LIN {X 0,Y 124.094,Z 764.223,A -85,B 0,C 180,E1 27360.319,E2 27360.319} C_VEL
LIN {X 0,Y 133.281,Z 757.884,A -85,B 0,C 180,E1 27361.4,E2 27361.4} C_VEL
LIN {X 0,Y 134.55,Z 756.801,A -85,B 0,C 180,E1 27362,E2 27362} C_VEL
LIN {X 0,Y 132.092,Z 757.455,A -85,B 0,C 180,E1 27366.547,E2 27366.547} C_VEL
LIN {X 0,Y 129.508,Z 758.725,A -85,B 0,C 180,E1 27369.46,E2 27369.46} C_VEL
LIN {X 0,Y 123.075,Z 762.693,A -85,B 0,C 180,E1 27371.274,E2 27371.274} C_VEL
LIN {X 0,Y 91.987,Z 778.369,A -85,B 0,C 180,E1 27378.553,E2 27378.553} C_VEL
LIN {X 0,Y 62.704,Z 788.454,A -85,B 0,C 180,E1 27392.644,E2 27392.644} C_VEL
LIN {X 0,Y 40.148,Z 793.378,A -85,B 0,C 180,E1 27427.943,E2 27427.943} C_VEL
LIN {X 0,Y 40.207,Z 793.347,A -85,B 0,C 180,E1 27472.061,E2 27472.061} C_VEL
LIN {X 0,Y 62.756,Z 788.368,A -85,B 0,C 180,E1 27507.325,E2 27507.325} C_VEL
LIN {X 0,Y 92.44,Z 778.051,A -85,B 0,C 180,E1 27521.5,E2 27521.5} C_VEL
LIN {X 0,Y 124.79,Z 761.469,A -85,B 0,C 180,E1 27528.95,E2 27528.95} C_VEL
LIN {X 0,Y 129.483,Z 758.548,A -85,B 0,C 180,E1 27530.56,E2 27530.56} C_VEL
LIN {X 0,Y 132.115,Z 757.233,A -85,B 0,C 180,E1 27533.454,E2 27533.454} C_VEL
LIN {X 0,Y 134.548,Z 756.597,A -85,B 0,C 180,E1 27538.001,E2 27538.001} C_VEL
LIN {X 0,Y 126.384,Z 762.482,A -85,B 0,C 180,E1 27539.383,E2 27539.383} C_VEL
LIN {X 0,Y 94.415,Z 781.112,A -85,B 0,C 180,E1 27544.833,E2 27544.833} C_VEL
LIN {X 0,Y 63.041,Z 794.367,A -85,B 0,C 180,E1 27556.741,E2 27556.741} C_VEL
LIN {X 0,Y 40.652,Z 801.7,A -85,B 0,C 180,E1 27582.041,E2 27582.041} C_VEL
LIN {X 0,Y 34.452,Z 804.774,A -85,B 0,C 180,E1 27629.345,E2 27629.345} C_VEL
LIN {X 0,Y 34.228,Z 804.663,A -85,B 0,C 180,E1 27643.351,E2 27643.351} C_VEL
LIN {X 0,Y 35.461,Z 800.565,A -85,B 0,C 180,E1 27687.235,E2 27687.235} C_VEL
LIN {X 0,Y 36.191,Z 800.352,A -85,B 0,C 180,E1 27688.651,E2 27688.651} C_VEL
LIN {X 0,Y 65.88,Z 791.602,A -85,B 0,C 180,E1 27712.667,E2 27712.667} C_VEL
LIN {X 0,Y 98.193,Z 777.913,A -85,B 0,C 180,E1 27720.886,E2 27720.886} C_VEL
LIN {X 0,Y 126.325,Z 761.604,A -85,B 0,C 180,E1 27724.614,E2 27724.614} C_VEL
LIN {X 0,Y 124.467,Z 762.35,A -85,B 0,C 180,E1 27726.95,E2 27726.95} C_VEL
LIN {X 0,Y 92.927,Z 778.287,A -85,B 0,C 180,E1 27733.062,E2 27733.062} C_VEL
LIN {X 0,Y 65.374,Z 787.866,A -85,B 0,C 180,E1 27742.624,E2 27742.624} C_VEL
LIN {X 0,Y 41.377,Z 793.304,A -85,B 0,C 180,E1 27763.193,E2 27763.193} C_VEL
LIN {X 0,Y 29.353,Z 795.095,A -85,B 0,C 180,E1 27810.025,E2 27810.025} C_VEL
LIN {X 0,Y 41.486,Z 793.244,A -85,B 0,C 180,E1 27856.698,E2 27856.698} C_VEL
LIN {X 0,Y 72.099,Z 785.77,A -85,B 0,C 180,E1 27880.383,E2 27880.383} C_VEL
LIN {X 0,Y 103.697,Z 773.349,A -85,B 0,C 180,E1 27889.212,E2 27889.212} C_VEL
LIN {X 0,Y 124.456,Z 762.164,A -85,B 0,C 180,E1 27893.05,E2 27893.05} C_VEL
LIN {X 0,Y 126.367,Z 761.386,A -85,B 0,C 180,E1 27895.382,E2 27895.382} C_VEL
LIN {X 0,Y 95.503,Z 779.134,A -85,B 0,C 180,E1 27899.572,E2 27899.572} C_VEL
LIN {X 0,Y 61.185,Z 793.12,A -85,B 0,C 180,E1 27909.364,E2 27909.364} C_VEL
LIN {X 0,Y 35.694,Z 800.457,A -85,B 0,C 180,E1 27932.24,E2 27932.24} C_VEL
LIN {X 0,Y 26.54,Z 803.586,A -85,B 0,C 180,E1 27989.973,E2 27989.973} C_VEL
LIN {X 0,Y 36.191,Z 800.352,A -85,B 0,C 180,E1 28048.651,E2 28048.651} C_VEL
LIN {X 0,Y 46.867,Z 796.623,A -85,B 0,C 180,E1 28067.322,E2 28067.322} C_VEL
LIN {X 0,Y 60.341,Z 791.95,A -85,B 0,C 180,E1 28078.38,E2 28078.38} C_VEL
LIN {X 0,Y 95.606,Z 778.16,A -85,B 0,C 180,E1 28085.323,E2 28085.323} C_VEL
LIN {X 0,Y 103.062,Z 774.499,A -85,B 0,C 180,E1 28086.079,E2 28086.079} C_VEL
LIN {X 0,Y 69.826,Z 787.065,A -85,B 0,C 180,E1 28093.53,E2 28093.53} C_VEL
LIN {X 0,Y 36.478,Z 794.49,A -85,B 0,C 180,E1 28114.212,E2 28114.212} C_VEL
LIN {X 0,Y 21.544,Z 796.282,A -85,B 0,C 180,E1 28170.034,E2 28170.034} C_VEL
LIN {X 0,Y 36.571,Z 794.431,A -85,B 0,C 180,E1 28225.644,E2 28225.644} C_VEL
LIN {X 0,Y 69.863,Z 786.962,A -85,B 0,C 180,E1 28246.435,E2 28246.435} C_VEL
LIN {X 0,Y 103.212,Z 774.29,A -85,B 0,C 180,E1 28253.914,E2 28253.914} C_VEL
LIN {X 0,Y 70.179,Z 788.574,A -85,B 0,C 180,E1 28258.944,E2 28258.944} C_VEL
LIN {X 0,Y 37.396,Z 798.04,A -85,B 0,C 180,E1 28273.988,E2 28273.988} C_VEL
LIN {X 0,Y 21.421,Z 801.316,A -85,B 0,C 180,E1 28305.17,E2 28305.17} C_VEL
LIN {X 0,Y 18.54,Z 802.371,A -85,B 0,C 180,E1 28349.961,E2 28349.961} C_VEL
LIN {X 0,Y 32.056,Z 799.249,A -85,B 0,C 180,E1 28420.225,E2 28420.225} C_VEL
LIN {X 0,Y 60.341,Z 791.95,A -85,B 0,C 180,E1 28438.38,E2 28438.38} C_VEL
LIN {X 0,Y 59.231,Z 791.67,A -85,B 0,C 180,E1 28442.189,E2 28442.189} C_VEL
LIN {X 0,Y 53.428,Z 792.556,A -85,B 0,C 180,E1 28446.947,E2 28446.947} C_VEL
LIN {X 0,Y 34.694,Z 795.461,A -85,B 0,C 180,E1 28461.032,E2 28461.032} C_VEL
LIN {X 0,Y 31.971,Z 795.746,A -85,B 0,C 180,E1 28463.533,E2 28463.533} C_VEL
LIN {X 0,Y 13.763,Z 797.464,A -85,B 0,C 180,E1 28530.053,E2 28530.053} C_VEL
LIN {X 0,Y 32.797,Z 795.62,A -85,B 0,C 180,E1 28597.006,E2 28597.006} C_VEL
LIN {X 0,Y 61.116,Z 790.16,A -85,B 0,C 180,E1 28611.036,E2 28611.036} C_VEL
LIN {X 0,Y 65.791,Z 789.027,A -85,B 0,C 180,E1 28612.984,E2 28612.984} C_VEL
LIN {X 0,Y 30.308,Z 797.97,A -85,B 0,C 180,E1 28625.039,E2 28625.039} C_VEL
LIN {X 0,Y 10.527,Z 801.154,A -85,B 0,C 180,E1 28709.931,E2 28709.931} C_VEL
LIN {X 0,Y 30.282,Z 798.006,A -85,B 0,C 180,E1 28794.973,E2 28794.973} C_VEL
LIN {X 0,Y 65.728,Z 789.134,A -85,B 0,C 180,E1 28807.007,E2 28807.007} C_VEL
LIN {X 0,Y 39.585,Z 794.659,A -85,B 0,C 180,E1 28817.704,E2 28817.704} C_VEL
LIN {X 0,Y 31.971,Z 795.746,A -85,B 0,C 180,E1 28823.533,E2 28823.533} C_VEL
LIN {X 0,Y 24.943,Z 796.903,A -85,B 0,C 180,E1 28824.135,E2 28824.135} C_VEL
LIN {X 0,Y 11.311,Z 799.26,A -85,B 0,C 180,E1 28801.153,E2 28801.153} C_VEL
LIN {X 0,Y 9.86,Z 799.371,A -85,B 0,C 180,E1 28798.609,E2 28798.609} C_VEL
LIN {X 0,Y 2.505,Z 799.935,A -85,B 0,C 180,E1 28709.709,E2 28709.709} C_VEL
LIN {X 0,Y 23.792,Z 797.786,A -85,B 0,C 180,E1 28611.393,E2 28611.393} C_VEL
LIN {X 0,Y 20.158,Z 797.842,A -85,B 0,C 180,E1 28603.349,E2 28603.349} C_VEL
LIN {X 0,Y 16.218,Z 798.123,A -85,B 0,C 180,E1 28461.626,E2 28461.626} C_VEL
LIN {X 0,Y 23.673,Z 797.839,A -85,B 0,C 180,E1 28448.557,E2 28448.557} C_VEL
LIN {X 0,Y 9.86,Z 799.371,A -85,B 0,C 180,E1 28438.609,E2 28438.609} C_VEL
LIN {X 0,Y 8.044,Z 801.368,A -85,B 0,C 180,E1 28435.281,E2 28435.281} C_VEL
LIN {X 0,Y 8.044,Z 875,A -85,B 0,C 180,E1 28435.281,E2 28435.281} C_VEL
LIN {X 0,Y 8.044,Z 875,A -85,B 0,C 180,E1 28435.281,E2 28435.281}

QRS_NEXT_CUT()
PTP {E1 28256.944,E2 28256.944}
PTP {X 0,Y 607.85,A -85,B 0,C 180,E1 28256.944,E2 28256.944,E3 0,E4 0,E5 0,E6 0}
QRS_SPEED_INIT()
LIN {X 0,Y 607.85,Z 875,A -85,B 0,C 180,E1 28256.944,E2 28256.944,E3 0,E4 0,E5 0,E6 0} C_VEL
LIN {X 0,Y 607.85,Z 296.842,A -85,B 0,C 180,E1 28256.944,E2 28256.944} C_VEL
LIN {X 0,Y 607.85,Z 288.764,A -85,B 0,C 180,E1 28256.944,E2 28256.944} C_VEL
LIN {X 0,Y 607.871,Z 286.764,A -85,B 0,C 180,E1 28256.755,E2 28256.755} C_VEL
LIN {X 0,Y 607.835,Z 286.764,A -85,B 0,C 180,E1 28253.672,E2 28253.672} C_VEL
LIN {X 0,Y 607.851,Z 286.764,A -85,B 0,C 180,E1 28250.914,E2 28250.914} C_VEL
LIN {X 0,Y 607.842,Z 286.764,A -85,B 0,C 180,E1 28247.652,E2 28247.652} C_VEL
LIN {X 0,Y 607.86,Z 286.764,A -85,B 0,C 180,E1 28244.839,E2 28244.839} C_VEL
LIN {X 0,Y 607.85,Z 286.762,A -85,B 0,C 180,E1 28241.589,E2 28241.589} C_VEL
LIN {X 0,Y 607.875,Z 286.764,A -85,B 0,C 180,E1 28238.684,E2 28238.684} C_VEL
LIN {X 0,Y 607.856,Z 286.761,A -85,B 0,C 180,E1 28235.511,E2 28235.511} C_VEL
LIN {X 0,Y 607.886,Z 286.764,A -85,B 0,C 180,E1 28232.577,E2 28232.577} C_VEL
LIN {X 0,Y 607.862,Z 286.761,A -85,B 0,C 180,E1 28229.451,E2 28229.451} C_VEL
LIN {X 0,Y 607.899,Z 286.764,A -85,B 0,C 180,E1 28226.451,E2 28226.451} C_VEL
LIN {X 0,Y 607.865,Z 286.76,A -85,B 0,C 180,E1 28223.338,E2 28223.338} C_VEL
LIN {X 0,Y 607.909,Z 286.765,A -85,B 0,C 180,E1 28220.329,E2 28220.329} C_VEL
LIN {X 0,Y 607.867,Z 286.76,A -85,B 0,C 180,E1 28217.188,E2 28217.188} C_VEL
LIN {X 0,Y 607.915,Z 286.761,A -85,B 0,C 180,E1 28214.083,E2 28214.083} C_VEL
LIN {X 0,Y 607.87,Z 286.76,A -85,B 0,C 180,E1 28210.975,E2 28210.975} C_VEL
LIN {X 0,Y 607.912,Z 286.759,A -85,B 0,C 180,E1 28207.841,E2 28207.841} C_VEL
LIN {X 0,Y 607.879,Z 286.761,A -85,B 0,C 180,E1 28204.687,E2 28204.687} C_VEL
LIN {X 0,Y 607.911,Z 286.755,A -85,B 0,C 180,E1 28201.535,E2 28201.535} C_VEL
LIN {X 0,Y 607.905,Z 286.765,A -85,B 0,C 180,E1 28198.273,E2 28198.273} C_VEL
LIN {X 0,Y 607.909,Z 287.028,A -85,B 0,C 180,E1 28196.259,E2 28196.259} C_VEL
LIN {X 0,Y 607.912,Z 319.926,A -85,B 0,C 180,E1 28193.454,E2 28193.454} C_VEL
LIN {X 0,Y 607.914,Z 334.281,A -85,B 0,C 180,E1 28192.278,E2 28192.278} C_VEL
LIN {X 0,Y 607.916,Z 541.958,A -85,B 0,C 180,E1 28189.666,E2 28189.666} C_VEL
LIN {X 0,Y 607.911,Z 560.928,A -85,B 0,C 180,E1 28189.25,E2 28189.25} C_VEL
LIN {X 0,Y 607.902,Z 579.266,A -85,B 0,C 180,E1 28188.668,E2 28188.668} C_VEL
LIN {X 0,Y 607.897,Z 597.163,A -85,B 0,C 180,E1 28187.913,E2 28187.913} C_VEL
LIN {X 0,Y 607.919,Z 613.869,A -85,B 0,C 180,E1 28187.023,E2 28187.023} C_VEL
LIN {X 0,Y 607.917,Z 629.704,A -85,B 0,C 180,E1 28185.991,E2 28185.991} C_VEL
LIN {X 0,Y 607.917,Z 644.611,A -85,B 0,C 180,E1 28184.818,E2 28184.818} C_VEL
LIN {X 0,Y 607.915,Z 658.52,A -85,B 0,C 180,E1 28183.506,E2 28183.506} C_VEL
LIN {X 0,Y 607.917,Z 671.323,A -85,B 0,C 180,E1 28182.056,E2 28182.056} C_VEL
LIN {X 0,Y 607.911,Z 682.566,A -85,B 0,C 180,E1 28180.519,E2 28180.519} C_VEL
LIN {X 0,Y 607.914,Z 692.264,A -85,B 0,C 180,E1 28178.894,E2 28178.894} C_VEL
LIN {X 0,Y 607.911,Z 699.987,A -85,B 0,C 180,E1 28177.276,E2 28177.276} C_VEL
LIN {X 0,Y 607.907,Z 706.267,A -85,B 0,C 180,E1 28175.569,E2 28175.569} C_VEL
LIN {X 0,Y 607.918,Z 710.775,A -85,B 0,C 180,E1 28173.867,E2 28173.867} C_VEL
LIN {X 0,Y 607.917,Z 713.734,A -85,B 0,C 180,E1 28172.074,E2 28172.074} C_VEL
LIN {X 0,Y 607.908,Z 714.929,A -85,B 0,C 180,E1 28170.283,E2 28170.283} C_VEL
LIN {X 0,Y 607.915,Z 714.38,A -85,B 0,C 180,E1 28168.492,E2 28168.492} C_VEL
LIN {X 0,Y 607.909,Z 712.08,A -85,B 0,C 180,E1 28166.7,E2 28166.7} C_VEL
LIN {X 0,Y 607.914,Z 708.217,A -85,B 0,C 180,E1 28164.999,E2 28164.999} C_VEL
LIN {X 0,Y 607.91,Z 702.635,A -85,B 0,C 180,E1 28163.294,E2 28163.294} C_VEL
LIN {X 0,Y 607.917,Z 695.641,A -85,B 0,C 180,E1 28161.678,E2 28161.678} C_VEL
LIN {X 0,Y 607.913,Z 686.781,A -85,B 0,C 180,E1 28160.056,E2 28160.056} C_VEL
LIN {X 0,Y 607.917,Z 676.477,A -85,B 0,C 180,E1 28158.521,E2 28158.521} C_VEL
LIN {X 0,Y 607.913,Z 664.743,A -85,B 0,C 180,E1 28157.075,E2 28157.075} C_VEL
LIN {X 0,Y 607.917,Z 651.561,A -85,B 0,C 180,E1 28155.718,E2 28155.718} C_VEL
LIN {X 0,Y 607.917,Z 636.801,A -85,B 0,C 180,E1 28154.45,E2 28154.45} C_VEL
LIN {X 0,Y 607.917,Z 620.944,A -85,B 0,C 180,E1 28153.322,E2 28153.322} C_VEL
LIN {X 0,Y 607.902,Z 603.949,A -85,B 0,C 180,E1 28152.335,E2 28152.335} C_VEL
LIN {X 0,Y 607.918,Z 586.961,A -85,B 0,C 180,E1 28151.543,E2 28151.543} C_VEL
LIN {X 0,Y 607.909,Z 569.084,A -85,B 0,C 180,E1 28150.895,E2 28150.895} C_VEL
LIN {X 0,Y 607.915,Z 550.763,A -85,B 0,C 180,E1 28150.413,E2 28150.413} C_VEL
LIN {X 0,Y 607.918,Z 531.813,A -85,B 0,C 180,E1 28150.096,E2 28150.096} C_VEL
LIN {X 0,Y 607.91,Z 334.059,A -85,B 0,C 180,E1 28147.621,E2 28147.621} C_VEL
LIN {X 0,Y 607.918,Z 296.429,A -85,B 0,C 180,E1 28144.475,E2 28144.475} C_VEL
LIN {X 0,Y 607.909,Z 286.947,A -85,B 0,C 180,E1 28143.636,E2 28143.636} C_VEL
LIN {X 0,Y 607.91,Z 286.756,A -85,B 0,C 180,E1 28140.543,E2 28140.543} C_VEL
LIN {X 0,Y 607.889,Z 286.762,A -85,B 0,C 180,E1 28137.352,E2 28137.352} C_VEL
LIN {X 0,Y 607.91,Z 286.758,A -85,B 0,C 180,E1 28134.181,E2 28134.181} C_VEL
LIN {X 0,Y 607.877,Z 286.76,A -85,B 0,C 180,E1 28131.075,E2 28131.075} C_VEL
LIN {X 0,Y 607.91,Z 286.76,A -85,B 0,C 180,E1 28127.98,E2 28127.98} C_VEL
LIN {X 0,Y 607.872,Z 286.759,A -85,B 0,C 180,E1 28124.882,E2 28124.882} C_VEL
LIN {X 0,Y 607.918,Z 286.764,A -85,B 0,C 180,E1 28121.696,E2 28121.696} C_VEL
LIN {X 0,Y 607.877,Z 286.759,A -85,B 0,C 180,E1 28118.565,E2 28118.565} C_VEL
LIN {X 0,Y 607.879,Z 286.763,A -85,B 0,C 180,E1 28115.264,E2 28115.264} C_VEL
LIN {X 0,Y 607.897,Z 286.758,A -85,B 0,C 180,E1 28112.203,E2 28112.203} C_VEL
LIN {X 0,Y 607.862,Z 286.762,A -85,B 0,C 180,E1 28109.028,E2 28109.028} C_VEL
LIN {X 0,Y 607.903,Z 286.759,A -85,B 0,C 180,E1 28106.05,E2 28106.05} C_VEL
LIN {X 0,Y 607.854,Z 286.763,A -85,B 0,C 180,E1 28102.91,E2 28102.91} C_VEL
LIN {X 0,Y 607.905,Z 286.76,A -85,B 0,C 180,E1 28099.905,E2 28099.905} C_VEL
LIN {X 0,Y 607.846,Z 286.763,A -85,B 0,C 180,E1 28096.801,E2 28096.801} C_VEL
LIN {X 0,Y 607.909,Z 286.761,A -85,B 0,C 180,E1 28093.798,E2 28093.798} C_VEL
LIN {X 0,Y 607.839,Z 286.764,A -85,B 0,C 180,E1 28090.713,E2 28090.713} C_VEL
LIN {X 0,Y 607.899,Z 286.762,A -85,B 0,C 180,E1 28087.751,E2 28087.751} C_VEL
LIN {X 0,Y 607.834,Z 286.764,A -85,B 0,C 180,E1 28084.718,E2 28084.718} C_VEL
LIN {X 0,Y 607.866,Z 286.764,A -85,B 0,C 180,E1 28081.885,E2 28081.885} C_VEL
LIN {X 0,Y 607.834,Z 286.765,A -85,B 0,C 180,E1 28078.775,E2 28078.775} C_VEL
LIN {X 0,Y 607.846,Z 286.764,A -85,B 0,C 180,E1 28076.039,E2 28076.039} C_VEL
LIN {X 0,Y 607.848,Z 286.763,A -85,B 0,C 180,E1 28072.819,E2 28072.819} C_VEL
LIN {X 0,Y 607.847,Z 286.764,A -85,B 0,C 180,E1 28070.054,E2 28070.054} C_VEL
LIN {X 0,Y 607.857,Z 286.762,A -85,B 0,C 180,E1 28066.783,E2 28066.783} C_VEL
LIN {X 0,Y 607.856,Z 286.764,A -85,B 0,C 180,E1 28063.958,E2 28063.958} C_VEL
LIN {X 0,Y 607.861,Z 286.761,A -85,B 0,C 180,E1 28060.694,E2 28060.694} C_VEL
LIN {X 0,Y 607.873,Z 286.764,A -85,B 0,C 180,E1 28057.771,E2 28057.771} C_VEL
LIN {X 0,Y 607.862,Z 286.761,A -85,B 0,C 180,E1 28054.557,E2 28054.557} C_VEL
LIN {X 0,Y 607.889,Z 286.764,A -85,B 0,C 180,E1 28051.618,E2 28051.618} C_VEL
LIN {X 0,Y 607.865,Z 286.76,A -85,B 0,C 180,E1 28048.432,E2 28048.432} C_VEL
LIN {X 0,Y 607.918,Z 286.763,A -85,B 0,C 180,E1 28045.314,E2 28045.314} C_VEL
LIN {X 0,Y 607.867,Z 286.76,A -85,B 0,C 180,E1 28042.274,E2 28042.274} C_VEL
LIN {X 0,Y 607.914,Z 286.761,A -85,B 0,C 180,E1 28039.162,E2 28039.162} C_VEL
LIN {X 0,Y 607.871,Z 286.76,A -85,B 0,C 180,E1 28036.042,E2 28036.042} C_VEL
LIN {X 0,Y 607.913,Z 286.759,A -85,B 0,C 180,E1 28032.914,E2 28032.914} C_VEL
LIN {X 0,Y 607.88,Z 286.761,A -85,B 0,C 180,E1 28029.778,E2 28029.778} C_VEL
LIN {X 0,Y 607.908,Z 286.756,A -85,B 0,C 180,E1 28026.54,E2 28026.54} C_VEL
LIN {X 0,Y 607.897,Z 286.884,A -85,B 0,C 180,E1 28023.498,E2 28023.498} C_VEL
LIN {X 0,Y 607.908,Z 287.709,A -85,B 0,C 180,E1 28023.382,E2 28023.382} C_VEL
LIN {X 0,Y 607.913,Z 340.141,A -85,B 0,C 180,E1 28020.435,E2 28020.435} C_VEL
LIN {X 0,Y 607.885,Z 390.509,A -85,B 0,C 180,E1 28017.701,E2 28017.701} C_VEL
LIN {X 0,Y 607.913,Z 616.116,A -85,B 0,C 180,E1 28014.784,E2 28014.784} C_VEL
LIN {X 0,Y 607.918,Z 653.733,A -85,B 0,C 180,E1 28014.278,E2 28014.278} C_VEL
LIN {X 0,Y 607.906,Z 673.698,A -85,B 0,C 180,E1 28013.84,E2 28013.84} C_VEL
LIN {X 0,Y 607.911,Z 693.06,A -85,B 0,C 180,E1 28013.249,E2 28013.249} C_VEL
LIN {X 0,Y 607.915,Z 712.501,A -85,B 0,C 180,E1 28012.482,E2 28012.482} C_VEL
LIN {X 0,Y 607.919,Z 731.168,A -85,B 0,C 180,E1 28011.567,E2 28011.567} C_VEL
LIN {X 0,Y 607.917,Z 749.766,A -85,B 0,C 180,E1 28010.456,E2 28010.456} C_VEL
LIN {X 0,Y 607.913,Z 767.254,A -85,B 0,C 180,E1 28009.204,E2 28009.204} C_VEL
LIN {X 0,Y 607.911,Z 783.162,A -85,B 0,C 180,E1 28007.863,E2 28007.863} C_VEL
LIN {X 0,Y 607.915,Z 797.673,A -85,B 0,C 180,E1 28006.432,E2 28006.432} C_VEL
LIN {X 0,Y 607.909,Z 811.263,A -85,B 0,C 180,E1 28004.867,E2 28004.867} C_VEL
LIN {X 0,Y 607.918,Z 823.719,A -85,B 0,C 180,E1 28003.176,E2 28003.176} C_VEL
LIN {X 0,Y 607.906,Z 834.252,A -85,B 0,C 180,E1 28001.479,E2 28001.479} C_VEL
LIN {X 0,Y 607.907,Z 843.561,A -85,B 0,C 180,E1 27999.658,E2 27999.658} C_VEL
LIN {X 0,Y 607.907,Z 850.973,A -85,B 0,C 180,E1 27997.846,E2 27997.846} C_VEL
LIN {X 0,Y 607.913,Z 856.989,A -85,B 0,C 180,E1 27995.947,E2 27995.947} C_VEL
LIN {X 0,Y 607.913,Z 861.292,A -85,B 0,C 180,E1 27994.055,E2 27994.055} C_VEL
LIN {X 0,Y 607.909,Z 863.95,A -85,B 0,C 180,E1 27992.168,E2 27992.168} C_VEL
LIN {X 0,Y 607.902,Z 864.94,A -85,B 0,C 180,E1 27990.283,E2 27990.283} C_VEL
LIN {X 0,Y 607.904,Z 864.372,A -85,B 0,C 180,E1 27988.398,E2 27988.398} C_VEL
LIN {X 0,Y 607.908,Z 862.082,A -85,B 0,C 180,E1 27986.417,E2 27986.417} C_VEL
LIN {X 0,Y 607.91,Z 858.255,A -85,B 0,C 180,E1 27984.526,E2 27984.526} C_VEL
LIN {X 0,Y 607.913,Z 852.689,A -85,B 0,C 180,E1 27982.629,E2 27982.629} C_VEL
LIN {X 0,Y 607.919,Z 845.655,A -85,B 0,C 180,E1 27980.82,E2 27980.82} C_VEL
LIN {X 0,Y 607.909,Z 836.843,A -85,B 0,C 180,E1 27979.001,E2 27979.001} C_VEL
LIN {X 0,Y 607.911,Z 826.516,A -85,B 0,C 180,E1 27977.247,E2 27977.247} C_VEL
LIN {X 0,Y 607.917,Z 815.136,A -85,B 0,C 180,E1 27975.62,E2 27975.62} C_VEL
LIN {X 0,Y 607.91,Z 801.355,A -85,B 0,C 180,E1 27973.96,E2 27973.96} C_VEL
LIN {X 0,Y 607.918,Z 785.904,A -85,B 0,C 180,E1 27972.385,E2 27972.385} C_VEL
LIN {X 0,Y 607.913,Z 769.201,A -85,B 0,C 180,E1 27970.945,E2 27970.945} C_VEL
LIN {X 0,Y 607.917,Z 752.006,A -85,B 0,C 180,E1 27969.694,E2 27969.694} C_VEL
LIN {X 0,Y 607.919,Z 734.735,A -85,B 0,C 180,E1 27968.636,E2 27968.636} C_VEL
LIN {X 0,Y 607.909,Z 715.856,A -85,B 0,C 180,E1 27967.671,E2 27967.671} C_VEL
LIN {X 0,Y 607.907,Z 696.731,A -85,B 0,C 180,E1 27966.879,E2 27966.879} C_VEL
LIN {X 0,Y 607.906,Z 676.741,A -85,B 0,C 180,E1 27966.237,E2 27966.237} C_VEL
LIN {X 0,Y 607.917,Z 657.663,A -85,B 0,C 180,E1 27965.799,E2 27965.799} C_VEL
LIN {X 0,Y 607.913,Z 631.428,A -85,B 0,C 180,E1 27965.411,E2 27965.411} C_VEL
LIN {X 0,Y 607.88,Z 396.039,A -85,B 0,C 180,E1 27962.375,E2 27962.375} C_VEL
LIN {X 0,Y 607.887,Z 389.594,A -85,B 0,C 180,E1 27962.26,E2 27962.26} C_VEL
LIN {X 0,Y 607.918,Z 333.456,A -85,B 0,C 180,E1 27959.195,E2 27959.195} C_VEL
LIN {X 0,Y 607.905,Z 287.421,A -85,B 0,C 180,E1 27956.592,E2 27956.592} C_VEL
LIN {X 0,Y 607.894,Z 286.812,A -85,B 0,C 180,E1 27956.452,E2 27956.452} C_VEL
LIN {X 0,Y 607.917,Z 286.756,A -85,B 0,C 180,E1 27953.343,E2 27953.343} C_VEL
LIN {X 0,Y 607.877,Z 286.76,A -85,B 0,C 180,E1 27950.099,E2 27950.099} C_VEL
LIN {X 0,Y 607.911,Z 286.761,A -85,B 0,C 180,E1 27946.957,E2 27946.957} C_VEL
LIN {X 0,Y 607.872,Z 286.76,A -85,B 0,C 180,E1 27943.827,E2 27943.827} C_VEL
LIN {X 0,Y 607.914,Z 286.765,A -85,B 0,C 180,E1 27940.641,E2 27940.641} C_VEL
LIN {X 0,Y 607.88,Z 286.758,A -85,B 0,C 180,E1 27937.487,E2 27937.487} C_VEL
LIN {X 0,Y 607.873,Z 286.763,A -85,B 0,C 180,E1 27934.174,E2 27934.174} C_VEL
LIN {X 0,Y 607.903,Z 286.758,A -85,B 0,C 180,E1 27931.095,E2 27931.095} C_VEL
LIN {X 0,Y 607.86,Z 286.762,A -85,B 0,C 180,E1 27927.956,E2 27927.956} C_VEL
LIN {X 0,Y 607.92,Z 286.759,A -85,B 0,C 180,E1 27924.901,E2 27924.901} C_VEL
LIN {X 0,Y 607.852,Z 286.762,A -85,B 0,C 180,E1 27921.823,E2 27921.823} C_VEL
LIN {X 0,Y 607.918,Z 286.762,A -85,B 0,C 180,E1 27918.706,E2 27918.706} C_VEL
LIN {X 0,Y 607.845,Z 286.763,A -85,B 0,C 180,E1 27915.65,E2 27915.65} C_VEL
LIN {X 0,Y 607.919,Z 286.764,A -85,B 0,C 180,E1 27912.539,E2 27912.539} C_VEL
LIN {X 0,Y 607.839,Z 286.763,A -85,B 0,C 180,E1 27909.563,E2 27909.563} C_VEL
LIN {X 0,Y 607.916,Z 286.764,A -85,B 0,C 180,E1 27906.516,E2 27906.516} C_VEL
LIN {X 0,Y 607.833,Z 286.764,A -85,B 0,C 180,E1 27903.489,E2 27903.489} C_VEL
LIN {X 0,Y 607.913,Z 286.765,A -85,B 0,C 180,E1 27900.471,E2 27900.471} C_VEL
LIN {X 0,Y 607.826,Z 286.765,A -85,B 0,C 180,E1 27897.454,E2 27897.454} C_VEL
LIN {X 0,Y 607.871,Z 286.764,A -85,B 0,C 180,E1 27896.755,E2 27896.755} C_VEL
LIN {X 0,Y 606.936,Z 286.888,A -85,B 0,C 180,E1 27896.029,E2 27896.029} C_VEL
LIN {X 0,Y 600.437,Z 287.691,A -85,B 0,C 180,E1 27893.992,E2 27893.992} C_VEL
LIN {X 0,Y 599.891,Z 287.754,A -85,B 0,C 180,E1 27893.462,E2 27893.462} C_VEL
LIN {X 0,Y 599.962,Z 287.753,A -85,B 0,C 180,E1 27890.503,E2 27890.503} C_VEL
LIN {X 0,Y 599.897,Z 287.753,A -85,B 0,C 180,E1 27887.486,E2 27887.486} C_VEL
LIN {X 0,Y 599.958,Z 287.752,A -85,B 0,C 180,E1 27884.535,E2 27884.535} C_VEL
LIN {X 0,Y 599.905,Z 287.751,A -85,B 0,C 180,E1 27881.437,E2 27881.437} C_VEL
LIN {X 0,Y 599.97,Z 287.754,A -85,B 0,C 180,E1 27878.389,E2 27878.389} C_VEL
LIN {X 0,Y 599.91,Z 287.75,A -85,B 0,C 180,E1 27875.27,E2 27875.27} C_VEL
LIN {X 0,Y 599.979,Z 287.75,A -85,B 0,C 180,E1 27872.185,E2 27872.185} C_VEL
LIN {X 0,Y 599.916,Z 287.751,A -85,B 0,C 180,E1 27869.114,E2 27869.114} C_VEL
LIN {X 0,Y 599.976,Z 287.749,A -85,B 0,C 180,E1 27866.063,E2 27866.063} C_VEL
LIN {X 0,Y 599.922,Z 287.751,A -85,B 0,C 180,E1 27862.968,E2 27862.968} C_VEL
LIN {X 0,Y 599.969,Z 287.747,A -85,B 0,C 180,E1 27859.838,E2 27859.838} C_VEL
LIN {X 0,Y 599.934,Z 287.751,A -85,B 0,C 180,E1 27856.743,E2 27856.743} C_VEL
LIN {X 0,Y 599.954,Z 287.745,A -85,B 0,C 180,E1 27853.493,E2 27853.493} C_VEL
LIN {X 0,Y 599.969,Z 287.755,A -85,B 0,C 180,E1 27850.285,E2 27850.285} C_VEL
LIN {X 0,Y 599.938,Z 287.748,A -85,B 0,C 180,E1 27847.106,E2 27847.106} C_VEL
LIN {X 0,Y 599.975,Z 287.752,A -85,B 0,C 180,E1 27844.051,E2 27844.051} C_VEL
LIN {X 0,Y 599.94,Z 287.748,A -85,B 0,C 180,E1 27840.874,E2 27840.874} C_VEL
LIN {X 0,Y 599.971,Z 287.752,A -85,B 0,C 180,E1 27837.707,E2 27837.707} C_VEL
LIN {X 0,Y 599.984,Z 288.004,A -85,B 0,C 180,E1 27836.553,E2 27836.553} C_VEL
LIN {X 0,Y 600.401,Z 291.081,A -85,B 0,C 180,E1 27836.24,E2 27836.24} C_VEL
LIN {X 0,Y 600.278,Z 327.914,A -85,B 0,C 180,E1 27833.095,E2 27833.095} C_VEL
LIN {X 0,Y 600.314,Z 334.297,A -85,B 0,C 180,E1 27832.575,E2 27832.575} C_VEL
LIN {X 0,Y 600.501,Z 346.221,A -85,B 0,C 180,E1 27832.404,E2 27832.404} C_VEL
LIN {X 0,Y 600.376,Z 542.325,A -85,B 0,C 180,E1 27829.917,E2 27829.917} C_VEL
LIN {X 0,Y 600.333,Z 561.284,A -85,B 0,C 180,E1 27829.493,E2 27829.493} C_VEL
LIN {X 0,Y 600.273,Z 579.732,A -85,B 0,C 180,E1 27828.896,E2 27828.896} C_VEL
LIN {X 0,Y 600.214,Z 597.173,A -85,B 0,C 180,E1 27828.15,E2 27828.15} C_VEL
LIN {X 0,Y 600.178,Z 613.876,A -85,B 0,C 180,E1 27827.249,E2 27827.249} C_VEL
LIN {X 0,Y 600.12,Z 629.709,A -85,B 0,C 180,E1 27826.204,E2 27826.204} C_VEL
LIN {X 0,Y 600.066,Z 644.618,A -85,B 0,C 180,E1 27825.016,E2 27825.016} C_VEL
LIN {X 0,Y 600.022,Z 658.526,A -85,B 0,C 180,E1 27823.687,E2 27823.687} C_VEL
LIN {X 0,Y 599.985,Z 671.33,A -85,B 0,C 180,E1 27822.218,E2 27822.218} C_VEL
LIN {X 0,Y 599.951,Z 682.571,A -85,B 0,C 180,E1 27820.66,E2 27820.66} C_VEL
LIN {X 0,Y 599.937,Z 692.268,A -85,B 0,C 180,E1 27819.013,E2 27819.013} C_VEL
LIN {X 0,Y 599.921,Z 699.99,A -85,B 0,C 180,E1 27817.373,E2 27817.373} C_VEL
LIN {X 0,Y 599.909,Z 706.269,A -85,B 0,C 180,E1 27815.643,E2 27815.643} C_VEL
LIN {X 0,Y 599.919,Z 710.778,A -85,B 0,C 180,E1 27813.918,E2 27813.918} C_VEL
LIN {X 0,Y 599.917,Z 713.736,A -85,B 0,C 180,E1 27812.101,E2 27812.101} C_VEL
LIN {X 0,Y 599.909,Z 714.929,A -85,B 0,C 180,E1 27810.286,E2 27810.286} C_VEL
LIN {X 0,Y 599.915,Z 714.38,A -85,B 0,C 180,E1 27808.472,E2 27808.472} C_VEL
LIN {X 0,Y 599.908,Z 712.08,A -85,B 0,C 180,E1 27806.656,E2 27806.656} C_VEL
LIN {X 0,Y 599.916,Z 708.216,A -85,B 0,C 180,E1 27804.932,E2 27804.932} C_VEL
LIN {X 0,Y 599.919,Z 702.634,A -85,B 0,C 180,E1 27803.204,E2 27803.204} C_VEL
LIN {X 0,Y 599.929,Z 695.639,A -85,B 0,C 180,E1 27801.567,E2 27801.567} C_VEL
LIN {X 0,Y 599.944,Z 686.779,A -85,B 0,C 180,E1 27799.922,E2 27799.922} C_VEL
LIN {X 0,Y 599.968,Z 676.473,A -85,B 0,C 180,E1 27798.367,E2 27798.367} C_VEL
LIN {X 0,Y 600,Z 664.738,A -85,B 0,C 180,E1 27796.901,E2 27796.901} C_VEL
LIN {X 0,Y 600.044,Z 651.243,A -85,B 0,C 180,E1 27795.496,E2 27795.496} C_VEL
LIN {X 0,Y 600.096,Z 636.79,A -85,B 0,C 180,E1 27794.242,E2 27794.242} C_VEL
LIN {X 0,Y 600.16,Z 620.933,A -85,B 0,C 180,E1 27793.1,E2 27793.1} C_VEL
LIN {X 0,Y 600.205,Z 603.942,A -85,B 0,C 180,E1 27792.101,E2 27792.101} C_VEL
LIN {X 0,Y 600.278,Z 586.855,A -85,B 0,C 180,E1 27791.295,E2 27791.295} C_VEL
LIN {X 0,Y 600.321,Z 568.317,A -85,B 0,C 180,E1 27790.622,E2 27790.622} C_VEL
LIN {X 0,Y 600.366,Z 549.69,A -85,B 0,C 180,E1 27790.136,E2 27790.136} C_VEL
LIN {X 0,Y 600.394,Z 529.98,A -85,B 0,C 180,E1 27789.813,E2 27789.813} C_VEL
LIN {X 0,Y 600.377,Z 334.753,A -85,B 0,C 180,E1 27787.35,E2 27787.35} C_VEL
LIN {X 0,Y 600.27,Z 329.595,A -85,B 0,C 180,E1 27786.957,E2 27786.957} C_VEL
LIN {X 0,Y 600.396,Z 292.735,A -85,B 0,C 180,E1 27783.813,E2 27783.813} C_VEL
LIN {X 0,Y 600.096,Z 288.551,A -85,B 0,C 180,E1 27783.431,E2 27783.431} C_VEL
LIN {X 0,Y 599.954,Z 287.79,A -85,B 0,C 180,E1 27783.259,E2 27783.259} C_VEL
LIN {X 0,Y 599.968,Z 287.751,A -85,B 0,C 180,E1 27780.065,E2 27780.065} C_VEL
LIN {X 0,Y 599.948,Z 287.747,A -85,B 0,C 180,E1 27776.865,E2 27776.865} C_VEL
LIN {X 0,Y 599.967,Z 287.753,A -85,B 0,C 180,E1 27773.604,E2 27773.604} C_VEL
LIN {X 0,Y 599.971,Z 287.744,A -85,B 0,C 180,E1 27770.338,E2 27770.338} C_VEL
LIN {X 0,Y 599.938,Z 287.748,A -85,B 0,C 180,E1 27767.16,E2 27767.16} C_VEL
LIN {X 0,Y 599.974,Z 287.747,A -85,B 0,C 180,E1 27764.022,E2 27764.022} C_VEL
LIN {X 0,Y 599.931,Z 287.749,A -85,B 0,C 180,E1 27760.919,E2 27760.919} C_VEL
LIN {X 0,Y 599.979,Z 287.753,A -85,B 0,C 180,E1 27757.706,E2 27757.706} C_VEL
LIN {X 0,Y 599.931,Z 287.748,A -85,B 0,C 180,E1 27754.585,E2 27754.585} C_VEL
LIN {X 0,Y 599.945,Z 287.752,A -85,B 0,C 180,E1 27751.331,E2 27751.331} C_VEL
LIN {X 0,Y 599.945,Z 287.748,A -85,B 0,C 180,E1 27748.25,E2 27748.25} C_VEL
LIN {X 0,Y 599.922,Z 287.751,A -85,B 0,C 180,E1 27745.045,E2 27745.045} C_VEL
LIN {X 0,Y 599.958,Z 287.749,A -85,B 0,C 180,E1 27742.023,E2 27742.023} C_VEL
LIN {X 0,Y 599.91,Z 287.752,A -85,B 0,C 180,E1 27738.865,E2 27738.865} C_VEL
LIN {X 0,Y 599.962,Z 287.75,A -85,B 0,C 180,E1 27735.862,E2 27735.862} C_VEL
LIN {X 0,Y 599.904,Z 287.752,A -85,B 0,C 180,E1 27732.807,E2 27732.807} C_VEL
LIN {X 0,Y 599.946,Z 287.751,A -85,B 0,C 180,E1 27729.884,E2 27729.884} C_VEL
LIN {X 0,Y 599.9,Z 287.753,A -85,B 0,C 180,E1 27726.796,E2 27726.796} C_VEL
LIN {X 0,Y 599.927,Z 287.753,A -85,B 0,C 180,E1 27723.918,E2 27723.918} C_VEL
LIN {X 0,Y 599.894,Z 287.754,A -85,B 0,C 180,E1 27720.764,E2 27720.764} C_VEL
LIN {X 0,Y 599.91,Z 287.753,A -85,B 0,C 180,E1 27717.994,E2 27717.994} C_VEL
LIN {X 0,Y 599.901,Z 287.753,A -85,B 0,C 180,E1 27714.741,E2 27714.741} C_VEL
LIN {X 0,Y 599.925,Z 287.753,A -85,B 0,C 180,E1 27711.856,E2 27711.856} C_VEL
LIN {X 0,Y 599.907,Z 287.752,A -85,B 0,C 180,E1 27708.658,E2 27708.658} C_VEL
LIN {X 0,Y 599.929,Z 287.752,A -85,B 0,C 180,E1 27705.819,E2 27705.819} C_VEL
LIN {X 0,Y 599.914,Z 287.751,A -85,B 0,C 180,E1 27702.643,E2 27702.643} C_VEL
LIN {X 0,Y 599.939,Z 287.753,A -85,B 0,C 180,E1 27699.717,E2 27699.717} C_VEL
LIN {X 0,Y 599.919,Z 287.75,A -85,B 0,C 180,E1 27696.526,E2 27696.526} C_VEL
LIN {X 0,Y 599.968,Z 287.754,A -85,B 0,C 180,E1 27693.473,E2 27693.473} C_VEL
LIN {X 0,Y 599.92,Z 287.75,A -85,B 0,C 180,E1 27690.331,E2 27690.331} C_VEL
LIN {X 0,Y 599.978,Z 287.751,A -85,B 0,C 180,E1 27687.207,E2 27687.207} C_VEL
LIN {X 0,Y 599.925,Z 287.748,A -85,B 0,C 180,E1 27684.08,E2 27684.08} C_VEL
LIN {X 0,Y 599.978,Z 287.747,A -85,B 0,C 180,E1 27680.947,E2 27680.947} C_VEL
LIN {X 0,Y 599.937,Z 287.748,A -85,B 0,C 180,E1 27677.806,E2 27677.806} C_VEL
LIN {X 0,Y 599.954,Z 287.745,A -85,B 0,C 180,E1 27674.497,E2 27674.497} C_VEL
LIN {X 0,Y 599.976,Z 287.753,A -85,B 0,C 180,E1 27671.272,E2 27671.272} C_VEL
LIN {X 0,Y 599.94,Z 287.749,A -85,B 0,C 180,E1 27668.07,E2 27668.07} C_VEL
LIN {X 0,Y 599.97,Z 287.745,A -85,B 0,C 180,E1 27664.923,E2 27664.923} C_VEL
LIN {X 0,Y 599.975,Z 287.98,A -85,B 0,C 180,E1 27663.91,E2 27663.91} C_VEL
LIN {X 0,Y 600.915,Z 290.689,A -85,B 0,C 180,E1 27663.646,E2 27663.646} C_VEL
LIN {X 0,Y 600.785,Z 342.119,A -85,B 0,C 180,E1 27660.725,E2 27660.725} C_VEL
LIN {X 0,Y 600.728,Z 391.1,A -85,B 0,C 180,E1 27658.048,E2 27658.048} C_VEL
LIN {X 0,Y 600.666,Z 596.888,A -85,B 0,C 180,E1 27655.353,E2 27655.353} C_VEL
LIN {X 0,Y 600.612,Z 654.257,A -85,B 0,C 180,E1 27654.583,E2 27654.583} C_VEL
LIN {X 0,Y 600.557,Z 674.736,A -85,B 0,C 180,E1 27654.124,E2 27654.124} C_VEL
LIN {X 0,Y 600.498,Z 693.797,A -85,B 0,C 180,E1 27653.527,E2 27653.527} C_VEL
LIN {X 0,Y 600.425,Z 713.624,A -85,B 0,C 180,E1 27652.726,E2 27652.726} C_VEL
LIN {X 0,Y 600.349,Z 732.065,A -85,B 0,C 180,E1 27651.801,E2 27651.801} C_VEL
LIN {X 0,Y 600.277,Z 750.54,A -85,B 0,C 180,E1 27650.678,E2 27650.678} C_VEL
LIN {X 0,Y 600.196,Z 768.576,A -85,B 0,C 180,E1 27649.36,E2 27649.36} C_VEL
LIN {X 0,Y 600.122,Z 785.371,A -85,B 0,C 180,E1 27647.902,E2 27647.902} C_VEL
LIN {X 0,Y 600.056,Z 800.903,A -85,B 0,C 180,E1 27646.307,E2 27646.307} C_VEL
LIN {X 0,Y 600.008,Z 814.366,A -85,B 0,C 180,E1 27644.672,E2 27644.672} C_VEL
LIN {X 0,Y 599.976,Z 826.017,A -85,B 0,C 180,E1 27643.001,E2 27643.001} C_VEL
LIN {X 0,Y 599.946,Z 836.327,A -85,B 0,C 180,E1 27641.244,E2 27641.244} C_VEL
LIN {X 0,Y 599.933,Z 845.34,A -85,B 0,C 180,E1 27639.378,E2 27639.378} C_VEL
LIN {X 0,Y 599.923,Z 852.38,A -85,B 0,C 180,E1 27637.566,E2 27637.566} C_VEL
LIN {X 0,Y 599.917,Z 858.002,A -85,B 0,C 180,E1 27635.643,E2 27635.643} C_VEL
LIN {X 0,Y 599.914,Z 861.924,A -85,B 0,C 180,E1 27633.727,E2 27633.727} C_VEL
LIN {X 0,Y 599.908,Z 864.306,A -85,B 0,C 180,E1 27631.719,E2 27631.719} C_VEL
LIN {X 0,Y 599.907,Z 864.962,A -85,B 0,C 180,E1 27629.809,E2 27629.809} C_VEL
LIN {X 0,Y 599.911,Z 864.039,A -85,B 0,C 180,E1 27627.899,E2 27627.899} C_VEL
LIN {X 0,Y 599.914,Z 861.451,A -85,B 0,C 180,E1 27625.986,E2 27625.986} C_VEL
LIN {X 0,Y 599.915,Z 857.242,A -85,B 0,C 180,E1 27624.069,E2 27624.069} C_VEL
LIN {X 0,Y 599.915,Z 851.327,A -85,B 0,C 180,E1 27622.145,E2 27622.145} C_VEL
LIN {X 0,Y 599.926,Z 844.017,A -85,B 0,C 180,E1 27620.31,E2 27620.31} C_VEL
LIN {X 0,Y 599.939,Z 834.772,A -85,B 0,C 180,E1 27618.464,E2 27618.464} C_VEL
LIN {X 0,Y 599.979,Z 824.098,A -85,B 0,C 180,E1 27616.705,E2 27616.705} C_VEL
LIN {X 0,Y 600.011,Z 812.04,A -85,B 0,C 180,E1 27615.032,E2 27615.032} C_VEL
LIN {X 0,Y 600.066,Z 798.599,A -85,B 0,C 180,E1 27613.446,E2 27613.446} C_VEL
LIN {X 0,Y 600.125,Z 783.715,A -85,B 0,C 180,E1 27611.948,E2 27611.948} C_VEL
LIN {X 0,Y 600.199,Z 767.851,A -85,B 0,C 180,E1 27610.584,E2 27610.584} C_VEL
LIN {X 0,Y 600.276,Z 750.539,A -85,B 0,C 180,E1 27609.322,E2 27609.322} C_VEL
LIN {X 0,Y 600.348,Z 732.063,A -85,B 0,C 180,E1 27608.199,E2 27608.199} C_VEL
LIN {X 0,Y 600.424,Z 713.621,A -85,B 0,C 180,E1 27607.274,E2 27607.274} C_VEL
LIN {X 0,Y 600.498,Z 693.796,A -85,B 0,C 180,E1 27606.473,E2 27606.473} C_VEL
LIN {X 0,Y 600.558,Z 674.063,A -85,B 0,C 180,E1 27605.859,E2 27605.859} C_VEL
LIN {X 0,Y 600.618,Z 653.731,A -85,B 0,C 180,E1 27605.407,E2 27605.407} C_VEL
LIN {X 0,Y 600.713,Z 509.726,A -85,B 0,C 180,E1 27603.515,E2 27603.515} C_VEL
LIN {X 0,Y 600.645,Z 390.371,A -85,B 0,C 180,E1 27601.932,E2 27601.932} C_VEL
LIN {X 0,Y 600.815,Z 334.206,A -85,B 0,C 180,E1 27598.832,E2 27598.832} C_VEL
LIN {X 0,Y 600.913,Z 290.688,A -85,B 0,C 180,E1 27596.354,E2 27596.354} C_VEL
LIN {X 0,Y 599.975,Z 287.98,A -85,B 0,C 180,E1 27596.09,E2 27596.09} C_VEL
LIN {X 0,Y 599.971,Z 287.749,A -85,B 0,C 180,E1 27593.016,E2 27593.016} C_VEL
LIN {X 0,Y 599.94,Z 287.747,A -85,B 0,C 180,E1 27589.838,E2 27589.838} C_VEL
LIN {X 0,Y 599.971,Z 287.751,A -85,B 0,C 180,E1 27586.602,E2 27586.602} C_VEL
LIN {X 0,Y 599.964,Z 287.746,A -85,B 0,C 180,E1 27583.362,E2 27583.362} C_VEL
LIN {X 0,Y 599.933,Z 287.751,A -85,B 0,C 180,E1 27580.097,E2 27580.097} C_VEL
LIN {X 0,Y 599.978,Z 287.747,A -85,B 0,C 180,E1 27576.985,E2 27576.985} C_VEL
LIN {X 0,Y 599.924,Z 287.75,A -85,B 0,C 180,E1 27573.825,E2 27573.825} C_VEL
LIN {X 0,Y 599.974,Z 287.753,A -85,B 0,C 180,E1 27570.66,E2 27570.66} C_VEL
LIN {X 0,Y 599.923,Z 287.749,A -85,B 0,C 180,E1 27567.547,E2 27567.547} C_VEL
LIN {X 0,Y 599.945,Z 287.752,A -85,B 0,C 180,E1 27564.308,E2 27564.308} C_VEL
LIN {X 0,Y 599.928,Z 287.75,A -85,B 0,C 180,E1 27561.304,E2 27561.304} C_VEL
LIN {X 0,Y 599.922,Z 287.752,A -85,B 0,C 180,E1 27558.059,E2 27558.059} C_VEL
LIN {X 0,Y 599.927,Z 287.751,A -85,B 0,C 180,E1 27555.168,E2 27555.168} C_VEL
LIN {X 0,Y 599.911,Z 287.753,A -85,B 0,C 180,E1 27551.927,E2 27551.927} C_VEL
LIN {X 0,Y 599.93,Z 287.751,A -85,B 0,C 180,E1 27549.013,E2 27549.013} C_VEL
LIN {X 0,Y 599.904,Z 287.753,A -85,B 0,C 180,E1 27545.835,E2 27545.835} C_VEL
LIN {X 0,Y 599.922,Z 287.752,A -85,B 0,C 180,E1 27542.961,E2 27542.961} C_VEL
LIN {X 0,Y 599.9,Z 287.754,A -85,B 0,C 180,E1 27539.809,E2 27539.809} C_VEL
LIN {X 0,Y 599.903,Z 287.753,A -85,B 0,C 180,E1 27537.038,E2 27537.038} C_VEL
LIN {X 0,Y 599.902,Z 287.753,A -85,B 0,C 180,E1 27533.78,E2 27533.78} C_VEL
LIN {X 0,Y 599.891,Z 287.754,A -85,B 0,C 180,E1 27533.462,E2 27533.462} C_VEL
LIN {X 0,Y 598.925,Z 287.88,A -85,B 0,C 180,E1 27532.726,E2 27532.726} C_VEL
LIN {X 0,Y 592.486,Z 288.687,A -85,B 0,C 180,E1 27530.608,E2 27530.608} C_VEL
LIN {X 0,Y 592.007,Z 288.741,A -85,B 0,C 180,E1 27530.125,E2 27530.125} C_VEL
LIN {X 0,Y 591.959,Z 288.742,A -85,B 0,C 180,E1 27527.216,E2 27527.216} C_VEL
LIN {X 0,Y 592.022,Z 288.74,A -85,B 0,C 180,E1 27524.121,E2 27524.121} C_VEL
LIN {X 0,Y 591.969,Z 288.741,A -85,B 0,C 180,E1 27521.077,E2 27521.077} C_VEL
LIN {X 0,Y 592.005,Z 288.739,A -85,B 0,C 180,E1 27517.874,E2 27517.874} C_VEL
LIN {X 0,Y 591.979,Z 288.739,A -85,B 0,C 180,E1 27514.916,E2 27514.916} C_VEL
LIN {X 0,Y 591.994,Z 288.738,A -85,B 0,C 180,E1 27511.633,E2 27511.633} C_VEL
LIN {X 0,Y 592,Z 288.741,A -85,B 0,C 180,E1 27508.654,E2 27508.654} C_VEL
LIN {X 0,Y 591.989,Z 288.738,A -85,B 0,C 180,E1 27505.424,E2 27505.424} C_VEL
LIN {X 0,Y 592.035,Z 288.742,A -85,B 0,C 180,E1 27502.312,E2 27502.312} C_VEL
LIN {X 0,Y 591.987,Z 288.738,A -85,B 0,C 180,E1 27499.169,E2 27499.169} C_VEL
LIN {X 0,Y 592.038,Z 288.737,A -85,B 0,C 180,E1 27496.007,E2 27496.007} C_VEL
LIN {X 0,Y 591.993,Z 288.736,A -85,B 0,C 180,E1 27492.86,E2 27492.86} C_VEL
LIN {X 0,Y 592.031,Z 288.733,A -85,B 0,C 180,E1 27489.635,E2 27489.635} C_VEL
LIN {X 0,Y 592.014,Z 288.741,A -85,B 0,C 180,E1 27486.476,E2 27486.476} C_VEL
LIN {X 0,Y 592.008,Z 288.736,A -85,B 0,C 180,E1 27483.175,E2 27483.175} C_VEL
LIN {X 0,Y 592.033,Z 288.742,A -85,B 0,C 180,E1 27479.959,E2 27479.959} C_VEL
LIN {X 0,Y 592.019,Z 288.846,A -85,B 0,C 180,E1 27476.907,E2 27476.907} C_VEL
LIN {X 0,Y 592.416,Z 290.475,A -85,B 0,C 180,E1 27476.675,E2 27476.675} C_VEL
LIN {X 0,Y 592.886,Z 293.544,A -85,B 0,C 180,E1 27476.382,E2 27476.382} C_VEL
LIN {X 0,Y 592.66,Z 329.764,A -85,B 0,C 180,E1 27473.251,E2 27473.251} C_VEL
LIN {X 0,Y 592.686,Z 334.316,A -85,B 0,C 180,E1 27472.882,E2 27472.882} C_VEL
LIN {X 0,Y 593.123,Z 338.906,A -85,B 0,C 180,E1 27472.792,E2 27472.792} C_VEL
LIN {X 0,Y 592.85,Z 542.359,A -85,B 0,C 180,E1 27470.181,E2 27470.181} C_VEL
LIN {X 0,Y 592.769,Z 561.326,A -85,B 0,C 180,E1 27469.752,E2 27469.752} C_VEL
LIN {X 0,Y 592.658,Z 579.704,A -85,B 0,C 180,E1 27469.15,E2 27469.15} C_VEL
LIN {X 0,Y 592.552,Z 597.183,A -85,B 0,C 180,E1 27468.393,E2 27468.393} C_VEL
LIN {X 0,Y 592.456,Z 613.883,A -85,B 0,C 180,E1 27467.481,E2 27467.481} C_VEL
LIN {X 0,Y 592.339,Z 629.714,A -85,B 0,C 180,E1 27466.423,E2 27466.423} C_VEL
LIN {X 0,Y 592.227,Z 644.624,A -85,B 0,C 180,E1 27465.22,E2 27465.22} C_VEL
LIN {X 0,Y 592.128,Z 658.532,A -85,B 0,C 180,E1 27463.873,E2 27463.873} C_VEL
LIN {X 0,Y 592.055,Z 671.336,A -85,B 0,C 180,E1 27462.384,E2 27462.384} C_VEL
LIN {X 0,Y 591.996,Z 682.577,A -85,B 0,C 180,E1 27460.805,E2 27460.805} C_VEL
LIN {X 0,Y 591.959,Z 692.273,A -85,B 0,C 180,E1 27459.135,E2 27459.135} C_VEL
LIN {X 0,Y 591.933,Z 700.036,A -85,B 0,C 180,E1 27457.463,E2 27457.463} C_VEL
LIN {X 0,Y 591.914,Z 706.272,A -85,B 0,C 180,E1 27455.72,E2 27455.72} C_VEL
LIN {X 0,Y 591.919,Z 710.78,A -85,B 0,C 180,E1 27453.971,E2 27453.971} C_VEL
LIN {X 0,Y 591.917,Z 713.737,A -85,B 0,C 180,E1 27452.13,E2 27452.13} C_VEL
LIN {X 0,Y 591.909,Z 714.929,A -85,B 0,C 180,E1 27450.29,E2 27450.29} C_VEL
LIN {X 0,Y 591.915,Z 714.38,A -85,B 0,C 180,E1 27448.451,E2 27448.451} C_VEL
LIN {X 0,Y 591.908,Z 712.08,A -85,B 0,C 180,E1 27446.611,E2 27446.611} C_VEL
LIN {X 0,Y 591.917,Z 708.215,A -85,B 0,C 180,E1 27444.864,E2 27444.864} C_VEL
LIN {X 0,Y 591.93,Z 702.632,A -85,B 0,C 180,E1 27443.112,E2 27443.112} C_VEL
LIN {X 0,Y 591.941,Z 695.636,A -85,B 0,C 180,E1 27441.452,E2 27441.452} C_VEL
LIN {X 0,Y 591.978,Z 686.777,A -85,B 0,C 180,E1 27439.785,E2 27439.785} C_VEL
LIN {X 0,Y 592.023,Z 676.47,A -85,B 0,C 180,E1 27438.209,E2 27438.209} C_VEL
LIN {X 0,Y 592.092,Z 664.733,A -85,B 0,C 180,E1 27436.723,E2 27436.723} C_VEL
LIN {X 0,Y 592.179,Z 651.547,A -85,B 0,C 180,E1 27435.33,E2 27435.33} C_VEL
LIN {X 0,Y 592.291,Z 636.779,A -85,B 0,C 180,E1 27434.029,E2 27434.029} C_VEL
LIN {X 0,Y 592.412,Z 620.92,A -85,B 0,C 180,E1 27432.872,E2 27432.872} C_VEL
LIN {X 0,Y 592.518,Z 603.836,A -85,B 0,C 180,E1 27431.856,E2 27431.856} C_VEL
LIN {X 0,Y 592.648,Z 586.494,A -85,B 0,C 180,E1 27431.031,E2 27431.031} C_VEL
LIN {X 0,Y 592.746,Z 568.083,A -85,B 0,C 180,E1 27430.358,E2 27430.358} C_VEL
LIN {X 0,Y 592.83,Z 549.495,A -85,B 0,C 180,E1 27429.87,E2 27429.87} C_VEL
LIN {X 0,Y 592.883,Z 529.801,A -85,B 0,C 180,E1 27429.545,E2 27429.545} C_VEL
LIN {X 0,Y 592.969,Z 335.979,A -85,B 0,C 180,E1 27427.074,E2 27427.074} C_VEL
LIN {X 0,Y 592.669,Z 334.111,A -85,B 0,C 180,E1 27427.017,E2 27427.017} C_VEL
LIN {X 0,Y 592.862,Z 297.641,A -85,B 0,C 180,E1 27423.886,E2 27423.886} C_VEL
LIN {X 0,Y 592.72,Z 291.498,A -85,B 0,C 180,E1 27423.34,E2 27423.34} C_VEL
LIN {X 0,Y 592.038,Z 288.941,A -85,B 0,C 180,E1 27423.041,E2 27423.041} C_VEL
LIN {X 0,Y 592.036,Z 288.74,A -85,B 0,C 180,E1 27419.848,E2 27419.848} C_VEL
LIN {X 0,Y 592.031,Z 288.734,A -85,B 0,C 180,E1 27416.543,E2 27416.543} C_VEL
LIN {X 0,Y 592.007,Z 288.74,A -85,B 0,C 180,E1 27413.283,E2 27413.283} C_VEL
LIN {X 0,Y 592.033,Z 288.735,A -85,B 0,C 180,E1 27410.063,E2 27410.063} C_VEL
LIN {X 0,Y 591.996,Z 288.735,A -85,B 0,C 180,E1 27406.975,E2 27406.975} C_VEL
LIN {X 0,Y 592.037,Z 288.739,A -85,B 0,C 180,E1 27403.823,E2 27403.823} C_VEL
LIN {X 0,Y 591.996,Z 288.737,A -85,B 0,C 180,E1 27400.684,E2 27400.684} C_VEL
LIN {X 0,Y 592.017,Z 288.742,A -85,B 0,C 180,E1 27397.446,E2 27397.446} C_VEL
LIN {X 0,Y 592.011,Z 288.736,A -85,B 0,C 180,E1 27394.325,E2 27394.325} C_VEL
LIN {X 0,Y 591.989,Z 288.74,A -85,B 0,C 180,E1 27391.098,E2 27391.098} C_VEL
LIN {X 0,Y 592.031,Z 288.736,A -85,B 0,C 180,E1 27388.002,E2 27388.002} C_VEL
LIN {X 0,Y 591.977,Z 288.738,A -85,B 0,C 180,E1 27384.871,E2 27384.871} C_VEL
LIN {X 0,Y 592.039,Z 288.74,A -85,B 0,C 180,E1 27381.746,E2 27381.746} C_VEL
LIN {X 0,Y 591.969,Z 288.74,A -85,B 0,C 180,E1 27378.644,E2 27378.644} C_VEL
LIN {X 0,Y 592.027,Z 288.741,A -85,B 0,C 180,E1 27375.477,E2 27375.477} C_VEL
LIN {X 0,Y 591.963,Z 288.741,A -85,B 0,C 180,E1 27372.486,E2 27372.486} C_VEL
LIN {X 0,Y 592.009,Z 288.74,A -85,B 0,C 180,E1 27369.331,E2 27369.331} C_VEL
LIN {X 0,Y 591.958,Z 288.742,A -85,B 0,C 180,E1 27366.401,E2 27366.401} C_VEL
LIN {X 0,Y 592.006,Z 288.741,A -85,B 0,C 180,E1 27363.292,E2 27363.292} C_VEL
LIN {X 0,Y 591.949,Z 288.743,A -85,B 0,C 180,E1 27360.387,E2 27360.387} C_VEL
LIN {X 0,Y 592.013,Z 288.741,A -85,B 0,C 180,E1 27357.29,E2 27357.29} C_VEL
LIN {X 0,Y 591.957,Z 288.742,A -85,B 0,C 180,E1 27354.281,E2 27354.281} C_VEL
LIN {X 0,Y 592.004,Z 288.74,A -85,B 0,C 180,E1 27351.115,E2 27351.115} C_VEL
LIN {X 0,Y 591.964,Z 288.742,A -85,B 0,C 180,E1 27348.207,E2 27348.207} C_VEL
LIN {X 0,Y 592.008,Z 288.74,A -85,B 0,C 180,E1 27345.025,E2 27345.025} C_VEL
LIN {X 0,Y 591.972,Z 288.741,A -85,B 0,C 180,E1 27342.097,E2 27342.097} C_VEL
LIN {X 0,Y 592.009,Z 288.738,A -85,B 0,C 180,E1 27338.916,E2 27338.916} C_VEL
LIN {X 0,Y 591.981,Z 288.74,A -85,B 0,C 180,E1 27335.981,E2 27335.981} C_VEL
LIN {X 0,Y 591.995,Z 288.737,A -85,B 0,C 180,E1 27332.652,E2 27332.652} C_VEL
LIN {X 0,Y 592.017,Z 288.742,A -85,B 0,C 180,E1 27329.558,E2 27329.558} C_VEL
LIN {X 0,Y 591.988,Z 288.738,A -85,B 0,C 180,E1 27326.359,E2 27326.359} C_VEL
LIN {X 0,Y 592.039,Z 288.738,A -85,B 0,C 180,E1 27323.284,E2 27323.284} C_VEL
LIN {X 0,Y 591.99,Z 288.739,A -85,B 0,C 180,E1 27320.065,E2 27320.065} C_VEL
LIN {X 0,Y 592.037,Z 288.737,A -85,B 0,C 180,E1 27316.977,E2 27316.977} C_VEL
LIN {X 0,Y 591.999,Z 288.738,A -85,B 0,C 180,E1 27313.824,E2 27313.824} C_VEL
LIN {X 0,Y 592.026,Z 288.732,A -85,B 0,C 180,E1 27310.537,E2 27310.537} C_VEL
LIN {X 0,Y 592.029,Z 288.739,A -85,B 0,C 180,E1 27307.302,E2 27307.302} C_VEL
LIN {X 0,Y 592.054,Z 288.974,A -85,B 0,C 180,E1 27304.365,E2 27304.365} C_VEL
LIN {X 0,Y 593.469,Z 292.667,A -85,B 0,C 180,E1 27304.009,E2 27304.009} C_VEL
LIN {X 0,Y 593.995,Z 294.645,A -85,B 0,C 180,E1 27303.859,E2 27303.859} C_VEL
LIN {X 0,Y 593.635,Z 348.076,A -85,B 0,C 180,E1 27300.797,E2 27300.797} C_VEL
LIN {X 0,Y 593.492,Z 391.113,A -85,B 0,C 180,E1 27298.421,E2 27298.421} C_VEL
LIN {X 0,Y 593.697,Z 408.263,A -85,B 0,C 180,E1 27298.179,E2 27298.179} C_VEL
LIN {X 0,Y 593.337,Z 653.628,A -85,B 0,C 180,E1 27294.917,E2 27294.917} C_VEL
LIN {X 0,Y 593.228,Z 673.971,A -85,B 0,C 180,E1 27294.461,E2 27294.461} C_VEL
LIN {X 0,Y 593.104,Z 693.8,A -85,B 0,C 180,E1 27293.838,E2 27293.838} C_VEL
LIN {X 0,Y 592.951,Z 713.627,A -85,B 0,C 180,E1 27293.029,E2 27293.029} C_VEL
LIN {X 0,Y 592.804,Z 732.062,A -85,B 0,C 180,E1 27292.093,E2 27292.093} C_VEL
LIN {X 0,Y 592.653,Z 750.537,A -85,B 0,C 180,E1 27290.956,E2 27290.956} C_VEL
LIN {X 0,Y 592.491,Z 768.577,A -85,B 0,C 180,E1 27289.622,E2 27289.622} C_VEL
LIN {X 0,Y 592.337,Z 785.5,A -85,B 0,C 180,E1 27288.133,E2 27288.133} C_VEL
LIN {X 0,Y 592.214,Z 800.453,A -85,B 0,C 180,E1 27286.578,E2 27286.578} C_VEL
LIN {X 0,Y 592.109,Z 813.592,A -85,B 0,C 180,E1 27284.972,E2 27284.972} C_VEL
LIN {X 0,Y 592.04,Z 825.379,A -85,B 0,C 180,E1 27283.278,E2 27283.278} C_VEL
LIN {X 0,Y 591.978,Z 836.328,A -85,B 0,C 180,E1 27281.397,E2 27281.397} C_VEL
LIN {X 0,Y 591.945,Z 845.249,A -85,B 0,C 180,E1 27279.528,E2 27279.528} C_VEL
LIN {X 0,Y 591.931,Z 852.38,A -85,B 0,C 180,E1 27277.668,E2 27277.668} C_VEL
LIN {X 0,Y 591.918,Z 858.002,A -85,B 0,C 180,E1 27275.72,E2 27275.72} C_VEL
LIN {X 0,Y 591.915,Z 861.925,A -85,B 0,C 180,E1 27273.777,E2 27273.777} C_VEL
LIN {X 0,Y 591.908,Z 864.307,A -85,B 0,C 180,E1 27271.742,E2 27271.742} C_VEL
LIN {X 0,Y 591.907,Z 864.962,A -85,B 0,C 180,E1 27269.806,E2 27269.806} C_VEL
LIN {X 0,Y 591.91,Z 864.038,A -85,B 0,C 180,E1 27267.87,E2 27267.87} C_VEL
LIN {X 0,Y 591.913,Z 861.451,A -85,B 0,C 180,E1 27265.932,E2 27265.932} C_VEL
LIN {X 0,Y 591.921,Z 857.243,A -85,B 0,C 180,E1 27263.989,E2 27263.989} C_VEL
LIN {X 0,Y 591.922,Z 851.328,A -85,B 0,C 180,E1 27262.038,E2 27262.038} C_VEL
LIN {X 0,Y 591.944,Z 844.017,A -85,B 0,C 180,E1 27260.178,E2 27260.178} C_VEL
LIN {X 0,Y 591.977,Z 834.773,A -85,B 0,C 180,E1 27258.306,E2 27258.306} C_VEL
LIN {X 0,Y 592.042,Z 824.099,A -85,B 0,C 180,E1 27256.523,E2 27256.523} C_VEL
LIN {X 0,Y 592.12,Z 812.041,A -85,B 0,C 180,E1 27254.827,E2 27254.827} C_VEL
LIN {X 0,Y 592.221,Z 798.333,A -85,B 0,C 180,E1 27253.191,E2 27253.191} C_VEL
LIN {X 0,Y 592.345,Z 783.715,A -85,B 0,C 180,E1 27251.702,E2 27251.702} C_VEL
LIN {X 0,Y 592.498,Z 767.944,A -85,B 0,C 180,E1 27250.329,E2 27250.329} C_VEL
LIN {X 0,Y 592.653,Z 750.536,A -85,B 0,C 180,E1 27249.044,E2 27249.044} C_VEL
LIN {X 0,Y 592.804,Z 732.06,A -85,B 0,C 180,E1 27247.907,E2 27247.907} C_VEL
LIN {X 0,Y 592.951,Z 713.624,A -85,B 0,C 180,E1 27246.971,E2 27246.971} C_VEL
LIN {X 0,Y 593.104,Z 693.798,A -85,B 0,C 180,E1 27246.161,E2 27246.161} C_VEL
LIN {X 0,Y 593.228,Z 673.972,A -85,B 0,C 180,E1 27245.539,E2 27245.539} C_VEL
LIN {X 0,Y 593.337,Z 653.731,A -85,B 0,C 180,E1 27245.085,E2 27245.085} C_VEL
LIN {X 0,Y 593.585,Z 495.247,A -85,B 0,C 180,E1 27242.979,E2 27242.979} C_VEL
LIN {X 0,Y 593.535,Z 391.421,A -85,B 0,C 180,E1 27241.586,E2 27241.586} C_VEL
LIN {X 0,Y 593.423,Z 386.627,A -85,B 0,C 180,E1 27241.358,E2 27241.358} C_VEL
LIN {X 0,Y 593.764,Z 330.25,A -85,B 0,C 180,E1 27238.193,E2 27238.193} C_VEL
LIN {X 0,Y 593.912,Z 293.959,A -85,B 0,C 180,E1 27236.096,E2 27236.096} C_VEL
LIN {X 0,Y 592.08,Z 289.145,A -85,B 0,C 180,E1 27235.666,E2 27235.666} C_VEL
LIN {X 0,Y 592.035,Z 288.729,A -85,B 0,C 180,E1 27235.311,E2 27235.311} C_VEL
LIN {X 0,Y 592.003,Z 288.741,A -85,B 0,C 180,E1 27232.188,E2 27232.188} C_VEL
LIN {X 0,Y 592.032,Z 288.736,A -85,B 0,C 180,E1 27229.018,E2 27229.018} C_VEL
LIN {X 0,Y 591.997,Z 288.736,A -85,B 0,C 180,E1 27225.873,E2 27225.873} C_VEL
LIN {X 0,Y 592.033,Z 288.74,A -85,B 0,C 180,E1 27222.724,E2 27222.724} C_VEL
LIN {X 0,Y 592.002,Z 288.737,A -85,B 0,C 180,E1 27219.548,E2 27219.548} C_VEL
LIN {X 0,Y 591.998,Z 288.737,A -85,B 0,C 180,E1 27216.237,E2 27216.237} C_VEL
LIN {X 0,Y 592.03,Z 288.736,A -85,B 0,C 180,E1 27213.107,E2 27213.107} C_VEL
LIN {X 0,Y 591.982,Z 288.74,A -85,B 0,C 180,E1 27209.884,E2 27209.884} C_VEL
LIN {X 0,Y 592.038,Z 288.738,A -85,B 0,C 180,E1 27206.803,E2 27206.803} C_VEL
LIN {X 0,Y 591.976,Z 288.739,A -85,B 0,C 180,E1 27203.702,E2 27203.702} C_VEL
LIN {X 0,Y 592.033,Z 288.744,A -85,B 0,C 180,E1 27200.566,E2 27200.566} C_VEL
LIN {X 0,Y 591.971,Z 288.74,A -85,B 0,C 180,E1 27197.496,E2 27197.496} C_VEL
LIN {X 0,Y 592.017,Z 288.74,A -85,B 0,C 180,E1 27194.375,E2 27194.375} C_VEL
LIN {X 0,Y 591.967,Z 288.741,A -85,B 0,C 180,E1 27191.398,E2 27191.398} C_VEL
LIN {X 0,Y 591.992,Z 288.741,A -85,B 0,C 180,E1 27188.156,E2 27188.156} C_VEL
LIN {X 0,Y 591.966,Z 288.742,A -85,B 0,C 180,E1 27185.233,E2 27185.233} C_VEL
LIN {X 0,Y 591.971,Z 288.742,A -85,B 0,C 180,E1 27181.936,E2 27181.936} C_VEL
LIN {X 0,Y 591.961,Z 288.743,A -85,B 0,C 180,E1 27179.129,E2 27179.129} C_VEL
LIN {X 0,Y 591.964,Z 288.742,A -85,B 0,C 180,E1 27175.835,E2 27175.835} C_VEL
LIN {X 0,Y 591.967,Z 288.743,A -85,B 0,C 180,E1 27173.015,E2 27173.015} C_VEL
LIN {X 0,Y 592.007,Z 288.741,A -85,B 0,C 180,E1 27170.125,E2 27170.125} C_VEL
LIN {X 0,Y 590.944,Z 288.872,A -85,B 0,C 180,E1 27169.379,E2 27169.379} C_VEL
LIN {X 0,Y 584.531,Z 289.669,A -85,B 0,C 180,E1 27167.288,E2 27167.288} C_VEL
LIN {X 0,Y 584.053,Z 289.731,A -85,B 0,C 180,E1 27166.743,E2 27166.743} C_VEL
LIN {X 0,Y 584.028,Z 289.73,A -85,B 0,C 180,E1 27163.489,E2 27163.489} C_VEL
LIN {X 0,Y 584.093,Z 289.729,A -85,B 0,C 180,E1 27160.396,E2 27160.396} C_VEL
LIN {X 0,Y 584.03,Z 289.73,A -85,B 0,C 180,E1 27157.237,E2 27157.237} C_VEL
LIN {X 0,Y 584.096,Z 289.728,A -85,B 0,C 180,E1 27154.118,E2 27154.118} C_VEL
LIN {X 0,Y 584.039,Z 289.729,A -85,B 0,C 180,E1 27151.02,E2 27151.02} C_VEL
LIN {X 0,Y 584.083,Z 289.726,A -85,B 0,C 180,E1 27147.833,E2 27147.833} C_VEL
LIN {X 0,Y 584.054,Z 289.73,A -85,B 0,C 180,E1 27144.743,E2 27144.743} C_VEL
LIN {X 0,Y 584.059,Z 289.726,A -85,B 0,C 180,E1 27141.454,E2 27141.454} C_VEL
LIN {X 0,Y 584.097,Z 289.73,A -85,B 0,C 180,E1 27138.249,E2 27138.249} C_VEL
LIN {X 0,Y 584.052,Z 289.726,A -85,B 0,C 180,E1 27135.006,E2 27135.006} C_VEL
LIN {X 0,Y 584.096,Z 289.727,A -85,B 0,C 180,E1 27131.872,E2 27131.872} C_VEL
LIN {X 0,Y 584.062,Z 289.727,A -85,B 0,C 180,E1 27128.669,E2 27128.669} C_VEL
LIN {X 0,Y 584.078,Z 289.723,A -85,B 0,C 180,E1 27125.352,E2 27125.352} C_VEL
LIN {X 0,Y 584.097,Z 289.728,A -85,B 0,C 180,E1 27122.076,E2 27122.076} C_VEL
LIN {X 0,Y 584.065,Z 289.73,A -85,B 0,C 180,E1 27118.865,E2 27118.865} C_VEL
LIN {X 0,Y 584.11,Z 289.95,A -85,B 0,C 180,E1 27117.196,E2 27117.196} C_VEL
LIN {X 0,Y 585.382,Z 295.394,A -85,B 0,C 180,E1 27116.583,E2 27116.583} C_VEL
LIN {X 0,Y 585.044,Z 331.749,A -85,B 0,C 180,E1 27113.4,E2 27113.4} C_VEL
LIN {X 0,Y 585.16,Z 334.92,A -85,B 0,C 180,E1 27113.179,E2 27113.179} C_VEL
LIN {X 0,Y 585.746,Z 339.839,A -85,B 0,C 180,E1 27113.084,E2 27113.084} C_VEL
LIN {X 0,Y 585.337,Z 542.393,A -85,B 0,C 180,E1 27110.452,E2 27110.452} C_VEL
LIN {X 0,Y 585.221,Z 561.393,A -85,B 0,C 180,E1 27110.016,E2 27110.016} C_VEL
LIN {X 0,Y 585.062,Z 579.718,A -85,B 0,C 180,E1 27109.409,E2 27109.409} C_VEL
LIN {X 0,Y 584.902,Z 597.193,A -85,B 0,C 180,E1 27108.642,E2 27108.642} C_VEL
LIN {X 0,Y 584.745,Z 613.89,A -85,B 0,C 180,E1 27107.719,E2 27107.719} C_VEL
LIN {X 0,Y 584.568,Z 629.719,A -85,B 0,C 180,E1 27106.648,E2 27106.648} C_VEL
LIN {X 0,Y 584.401,Z 644.602,A -85,B 0,C 180,E1 27105.431,E2 27105.431} C_VEL
LIN {X 0,Y 584.248,Z 658.538,A -85,B 0,C 180,E1 27104.064,E2 27104.064} C_VEL
LIN {X 0,Y 584.131,Z 671.343,A -85,B 0,C 180,E1 27102.555,E2 27102.555} C_VEL
LIN {X 0,Y 584.043,Z 682.582,A -85,B 0,C 180,E1 27100.954,E2 27100.954} C_VEL
LIN {X 0,Y 583.984,Z 692.278,A -85,B 0,C 180,E1 27099.261,E2 27099.261} C_VEL
LIN {X 0,Y 583.945,Z 700.219,A -85,B 0,C 180,E1 27097.521,E2 27097.521} C_VEL
LIN {X 0,Y 583.917,Z 706.275,A -85,B 0,C 180,E1 27095.798,E2 27095.798} C_VEL
LIN {X 0,Y 583.919,Z 710.782,A -85,B 0,C 180,E1 27094.026,E2 27094.026} C_VEL
LIN {X 0,Y 583.916,Z 713.739,A -85,B 0,C 180,E1 27092.159,E2 27092.159} C_VEL
LIN {X 0,Y 583.909,Z 714.929,A -85,B 0,C 180,E1 27090.294,E2 27090.294} C_VEL
LIN {X 0,Y 583.914,Z 714.38,A -85,B 0,C 180,E1 27088.43,E2 27088.43} C_VEL
LIN {X 0,Y 583.908,Z 712.079,A -85,B 0,C 180,E1 27086.564,E2 27086.564} C_VEL
LIN {X 0,Y 583.919,Z 708.214,A -85,B 0,C 180,E1 27084.793,E2 27084.793} C_VEL
LIN {X 0,Y 583.938,Z 702.63,A -85,B 0,C 180,E1 27083.017,E2 27083.017} C_VEL
LIN {X 0,Y 583.956,Z 695.634,A -85,B 0,C 180,E1 27081.334,E2 27081.334} C_VEL
LIN {X 0,Y 584.014,Z 686.774,A -85,B 0,C 180,E1 27079.644,E2 27079.644} C_VEL
LIN {X 0,Y 584.083,Z 676.467,A -85,B 0,C 180,E1 27078.046,E2 27078.046} C_VEL
LIN {X 0,Y 584.19,Z 664.728,A -85,B 0,C 180,E1 27076.54,E2 27076.54} C_VEL
LIN {X 0,Y 584.326,Z 651.539,A -85,B 0,C 180,E1 27075.128,E2 27075.128} C_VEL
LIN {X 0,Y 584.491,Z 636.768,A -85,B 0,C 180,E1 27073.81,E2 27073.81} C_VEL
LIN {X 0,Y 584.673,Z 620.906,A -85,B 0,C 180,E1 27072.638,E2 27072.638} C_VEL
LIN {X 0,Y 584.841,Z 603.926,A -85,B 0,C 180,E1 27071.614,E2 27071.614} C_VEL
LIN {X 0,Y 585.026,Z 586.92,A -85,B 0,C 180,E1 27070.793,E2 27070.793} C_VEL
LIN {X 0,Y 585.179,Z 568.39,A -85,B 0,C 180,E1 27070.103,E2 27070.103} C_VEL
LIN {X 0,Y 585.306,Z 549.625,A -85,B 0,C 180,E1 27069.603,E2 27069.603} C_VEL
LIN {X 0,Y 585.385,Z 529.877,A -85,B 0,C 180,E1 27069.272,E2 27069.272} C_VEL
LIN {X 0,Y 585.591,Z 337.201,A -85,B 0,C 180,E1 27066.785,E2 27066.785} C_VEL
LIN {X 0,Y 585.049,Z 334.004,A -85,B 0,C 180,E1 27066.695,E2 27066.695} C_VEL
LIN {X 0,Y 585.363,Z 297.512,A -85,B 0,C 180,E1 27063.515,E2 27063.515} C_VEL
LIN {X 0,Y 585.222,Z 293.947,A -85,B 0,C 180,E1 27063.19,E2 27063.19} C_VEL
LIN {X 0,Y 584.111,Z 289.888,A -85,B 0,C 180,E1 27062.694,E2 27062.694} C_VEL
LIN {X 0,Y 584.073,Z 289.725,A -85,B 0,C 180,E1 27059.328,E2 27059.328} C_VEL
LIN {X 0,Y 584.092,Z 289.727,A -85,B 0,C 180,E1 27056.08,E2 27056.08} C_VEL
LIN {X 0,Y 584.064,Z 289.726,A -85,B 0,C 180,E1 27052.916,E2 27052.916} C_VEL
LIN {X 0,Y 584.094,Z 289.732,A -85,B 0,C 180,E1 27049.62,E2 27049.62} C_VEL
LIN {X 0,Y 584.089,Z 289.719,A -85,B 0,C 180,E1 27046.382,E2 27046.382} C_VEL
LIN {X 0,Y 584.061,Z 289.729,A -85,B 0,C 180,E1 27043.176,E2 27043.176} C_VEL
LIN {X 0,Y 584.098,Z 289.725,A -85,B 0,C 180,E1 27040.064,E2 27040.064} C_VEL
LIN {X 0,Y 584.05,Z 289.728,A -85,B 0,C 180,E1 27036.922,E2 27036.922} C_VEL
LIN {X 0,Y 584.099,Z 289.729,A -85,B 0,C 180,E1 27033.705,E2 27033.705} C_VEL
LIN {X 0,Y 584.05,Z 289.727,A -85,B 0,C 180,E1 27030.561,E2 27030.561} C_VEL
LIN {X 0,Y 584.065,Z 289.731,A -85,B 0,C 180,E1 27027.309,E2 27027.309} C_VEL
LIN {X 0,Y 584.059,Z 289.725,A -85,B 0,C 180,E1 27024.259,E2 27024.259} C_VEL
LIN {X 0,Y 584.04,Z 289.729,A -85,B 0,C 180,E1 27020.965,E2 27020.965} C_VEL
LIN {X 0,Y 584.091,Z 289.727,A -85,B 0,C 180,E1 27017.844,E2 27017.844} C_VEL
LIN {X 0,Y 584.027,Z 289.727,A -85,B 0,C 180,E1 27014.678,E2 27014.678} C_VEL
LIN {X 0,Y 584.096,Z 289.732,A -85,B 0,C 180,E1 27011.554,E2 27011.554} C_VEL
LIN {X 0,Y 584.021,Z 289.727,A -85,B 0,C 180,E1 27008.467,E2 27008.467} C_VEL
LIN {X 0,Y 584.068,Z 289.731,A -85,B 0,C 180,E1 27005.304,E2 27005.304} C_VEL
LIN {X 0,Y 584.015,Z 289.729,A -85,B 0,C 180,E1 27002.355,E2 27002.355} C_VEL
LIN {X 0,Y 584.058,Z 289.731,A -85,B 0,C 180,E1 26999.215,E2 26999.215} C_VEL
LIN {X 0,Y 584.016,Z 289.73,A -85,B 0,C 180,E1 26996.27,E2 26996.27} C_VEL
LIN {X 0,Y 584.06,Z 289.729,A -85,B 0,C 180,E1 26993.118,E2 26993.118} C_VEL
LIN {X 0,Y 584.026,Z 289.73,A -85,B 0,C 180,E1 26990.143,E2 26990.143} C_VEL
LIN {X 0,Y 584.045,Z 289.726,A -85,B 0,C 180,E1 26986.839,E2 26986.839} C_VEL
LIN {X 0,Y 584.045,Z 289.731,A -85,B 0,C 180,E1 26983.899,E2 26983.899} C_VEL
LIN {X 0,Y 584.04,Z 289.728,A -85,B 0,C 180,E1 26980.603,E2 26980.603} C_VEL
LIN {X 0,Y 584.08,Z 289.731,A -85,B 0,C 180,E1 26977.559,E2 26977.559} C_VEL
LIN {X 0,Y 584.038,Z 289.729,A -85,B 0,C 180,E1 26974.334,E2 26974.334} C_VEL
LIN {X 0,Y 584.102,Z 289.729,A -85,B 0,C 180,E1 26971.212,E2 26971.212} C_VEL
LIN {X 0,Y 584.045,Z 289.728,A -85,B 0,C 180,E1 26968.063,E2 26968.063} C_VEL
LIN {X 0,Y 584.094,Z 289.719,A -85,B 0,C 180,E1 26964.889,E2 26964.889} C_VEL
LIN {X 0,Y 584.064,Z 289.729,A -85,B 0,C 180,E1 26961.705,E2 26961.705} C_VEL
LIN {X 0,Y 584.061,Z 289.719,A -85,B 0,C 180,E1 26958.378,E2 26958.378} C_VEL
LIN {X 0,Y 584.099,Z 289.729,A -85,B 0,C 180,E1 26955.265,E2 26955.265} C_VEL
LIN {X 0,Y 584.058,Z 289.728,A -85,B 0,C 180,E1 26952.015,E2 26952.015} C_VEL
LIN {X 0,Y 584.096,Z 289.728,A -85,B 0,C 180,E1 26948.843,E2 26948.843} C_VEL
LIN {X 0,Y 584.075,Z 289.734,A -85,B 0,C 180,E1 26945.593,E2 26945.593} C_VEL
LIN {X 0,Y 584.139,Z 290.034,A -85,B 0,C 180,E1 26944.823,E2 26944.823} C_VEL
LIN {X 0,Y 587.056,Z 297.689,A -85,B 0,C 180,E1 26944.133,E2 26944.133} C_VEL
LIN {X 0,Y 586.515,Z 351.021,A -85,B 0,C 180,E1 26941.042,E2 26941.042} C_VEL
LIN {X 0,Y 586.276,Z 391.086,A -85,B 0,C 180,E1 26938.804,E2 26938.804} C_VEL
LIN {X 0,Y 586.677,Z 397.066,A -85,B 0,C 180,E1 26938.7,E2 26938.7} C_VEL
LIN {X 0,Y 586.142,Z 631.431,A -85,B 0,C 180,E1 26935.567,E2 26935.567} C_VEL
LIN {X 0,Y 586.031,Z 658.151,A -85,B 0,C 180,E1 26935.156,E2 26935.156} C_VEL
LIN {X 0,Y 585.863,Z 678.255,A -85,B 0,C 180,E1 26934.669,E2 26934.669} C_VEL
LIN {X 0,Y 585.699,Z 698.068,A -85,B 0,C 180,E1 26934.003,E2 26934.003} C_VEL
LIN {X 0,Y 585.469,Z 716.988,A -85,B 0,C 180,E1 26933.181,E2 26933.181} C_VEL
LIN {X 0,Y 585.221,Z 735.717,A -85,B 0,C 180,E1 26932.178,E2 26932.178} C_VEL
LIN {X 0,Y 584.966,Z 754.196,A -85,B 0,C 180,E1 26930.982,E2 26930.982} C_VEL
LIN {X 0,Y 584.73,Z 771.625,A -85,B 0,C 180,E1 26929.633,E2 26929.633} C_VEL
LIN {X 0,Y 584.524,Z 787.62,A -85,B 0,C 180,E1 26928.17,E2 26928.17} C_VEL
LIN {X 0,Y 584.348,Z 802.207,A -85,B 0,C 180,E1 26926.603,E2 26926.603} C_VEL
LIN {X 0,Y 584.197,Z 815.861,A -85,B 0,C 180,E1 26924.875,E2 26924.875} C_VEL
LIN {X 0,Y 584.091,Z 827.93,A -85,B 0,C 180,E1 26923.059,E2 26923.059} C_VEL
LIN {X 0,Y 584.005,Z 838.399,A -85,B 0,C 180,E1 26921.155,E2 26921.155} C_VEL
LIN {X 0,Y 583.962,Z 846.875,A -85,B 0,C 180,E1 26919.262,E2 26919.262} C_VEL
LIN {X 0,Y 583.93,Z 853.9,A -85,B 0,C 180,E1 26917.279,E2 26917.279} C_VEL
LIN {X 0,Y 583.914,Z 859.144,A -85,B 0,C 180,E1 26915.305,E2 26915.305} C_VEL
LIN {X 0,Y 583.909,Z 862.71,A -85,B 0,C 180,E1 26913.338,E2 26913.338} C_VEL
LIN {X 0,Y 583.905,Z 864.639,A -85,B 0,C 180,E1 26911.275,E2 26911.275} C_VEL
LIN {X 0,Y 583.904,Z 864.851,A -85,B 0,C 180,E1 26909.313,E2 26909.313} C_VEL
LIN {X 0,Y 583.91,Z 863.392,A -85,B 0,C 180,E1 26907.252,E2 26907.252} C_VEL
LIN {X 0,Y 583.918,Z 860.169,A -85,B 0,C 180,E1 26905.187,E2 26905.187} C_VEL
LIN {X 0,Y 583.931,Z 855.414,A -85,B 0,C 180,E1 26903.215,E2 26903.215} C_VEL
LIN {X 0,Y 583.948,Z 848.851,A -85,B 0,C 180,E1 26901.235,E2 26901.235} C_VEL
LIN {X 0,Y 583.98,Z 840.795,A -85,B 0,C 180,E1 26899.344,E2 26899.344} C_VEL
LIN {X 0,Y 584.05,Z 830.838,A -85,B 0,C 180,E1 26897.443,E2 26897.443} C_VEL
LIN {X 0,Y 584.159,Z 819.391,A -85,B 0,C 180,E1 26895.63,E2 26895.63} C_VEL
LIN {X 0,Y 584.299,Z 806.451,A -85,B 0,C 180,E1 26893.906,E2 26893.906} C_VEL
LIN {X 0,Y 584.476,Z 791.978,A -85,B 0,C 180,E1 26892.272,E2 26892.272} C_VEL
LIN {X 0,Y 584.683,Z 776.45,A -85,B 0,C 180,E1 26890.781,E2 26890.781} C_VEL
LIN {X 0,Y 584.922,Z 759.28,A -85,B 0,C 180,E1 26889.383,E2 26889.383} C_VEL
LIN {X 0,Y 585.174,Z 740.916,A -85,B 0,C 180,E1 26888.132,E2 26888.132} C_VEL
LIN {X 0,Y 585.388,Z 722.299,A -85,B 0,C 180,E1 26887.082,E2 26887.082} C_VEL
LIN {X 0,Y 585.612,Z 702.731,A -85,B 0,C 180,E1 26886.185,E2 26886.185} C_VEL
LIN {X 0,Y 585.833,Z 682.304,A -85,B 0,C 180,E1 26885.456,E2 26885.456} C_VEL
LIN {X 0,Y 586.013,Z 662.109,A -85,B 0,C 180,E1 26884.925,E2 26884.925} C_VEL
LIN {X 0,Y 586.122,Z 641.479,A -85,B 0,C 180,E1 26884.566,E2 26884.566} C_VEL
LIN {X 0,Y 586.657,Z 403.425,A -85,B 0,C 180,E1 26881.386,E2 26881.386} C_VEL
LIN {X 0,Y 586.434,Z 392.169,A -85,B 0,C 180,E1 26881.22,E2 26881.22} C_VEL
LIN {X 0,Y 586.183,Z 389.594,A -85,B 0,C 180,E1 26881.138,E2 26881.138} C_VEL
LIN {X 0,Y 586.704,Z 333.118,A -85,B 0,C 180,E1 26877.932,E2 26877.932} C_VEL
LIN {X 0,Y 586.959,Z 297.044,A -85,B 0,C 180,E1 26875.822,E2 26875.822} C_VEL
LIN {X 0,Y 584.146,Z 290.078,A -85,B 0,C 180,E1 26875.182,E2 26875.182} C_VEL
LIN {X 0,Y 584.087,Z 289.73,A -85,B 0,C 180,E1 26874.57,E2 26874.57} C_VEL
LIN {X 0,Y 584.096,Z 289.726,A -85,B 0,C 180,E1 26871.314,E2 26871.314} C_VEL
LIN {X 0,Y 584.061,Z 289.729,A -85,B 0,C 180,E1 26868.116,E2 26868.116} C_VEL
LIN {X 0,Y 584.097,Z 289.726,A -85,B 0,C 180,E1 26864.874,E2 26864.874} C_VEL
LIN {X 0,Y 584.057,Z 289.719,A -85,B 0,C 180,E1 26861.723,E2 26861.723} C_VEL
LIN {X 0,Y 584.077,Z 289.729,A -85,B 0,C 180,E1 26858.419,E2 26858.419} C_VEL
LIN {X 0,Y 584.083,Z 289.719,A -85,B 0,C 180,E1 26855.232,E2 26855.232} C_VEL
LIN {X 0,Y 584.05,Z 289.729,A -85,B 0,C 180,E1 26852.053,E2 26852.053} C_VEL
LIN {X 0,Y 584.098,Z 289.728,A -85,B 0,C 180,E1 26848.863,E2 26848.863} C_VEL
LIN {X 0,Y 584.039,Z 289.729,A -85,B 0,C 180,E1 26845.775,E2 26845.775} C_VEL
LIN {X 0,Y 584.102,Z 289.728,A -85,B 0,C 180,E1 26842.653,E2 26842.653} C_VEL
LIN {X 0,Y 584.037,Z 289.728,A -85,B 0,C 180,E1 26839.502,E2 26839.502} C_VEL
LIN {X 0,Y 584.069,Z 289.731,A -85,B 0,C 180,E1 26836.305,E2 26836.305} C_VEL
LIN {X 0,Y 584.033,Z 289.726,A -85,B 0,C 180,E1 26833.363,E2 26833.363} C_VEL
LIN {X 0,Y 584.043,Z 289.73,A -85,B 0,C 180,E1 26830.056,E2 26830.056} C_VEL
LIN {X 0,Y 584.034,Z 289.728,A -85,B 0,C 180,E1 26827.179,E2 26827.179} C_VEL
LIN {X 0,Y 584.025,Z 289.73,A -85,B 0,C 180,E1 26823.828,E2 26823.828} C_VEL
LIN {X 0,Y 584.048,Z 289.73,A -85,B 0,C 180,E1 26820.883,E2 26820.883} C_VEL
LIN {X 0,Y 584.013,Z 289.73,A -85,B 0,C 180,E1 26817.645,E2 26817.645} C_VEL
LIN {X 0,Y 584.073,Z 289.731,A -85,B 0,C 180,E1 26814.597,E2 26814.597} C_VEL
LIN {X 0,Y 584.017,Z 289.728,A -85,B 0,C 180,E1 26811.533,E2 26811.533} C_VEL
LIN {X 0,Y 584.09,Z 289.732,A -85,B 0,C 180,E1 26808.446,E2 26808.446} C_VEL
LIN {X 0,Y 584.053,Z 289.731,A -85,B 0,C 180,E1 26806.743,E2 26806.743} C_VEL
LIN {X 0,Y 583.114,Z 289.855,A -85,B 0,C 180,E1 26805.987,E2 26805.987} C_VEL
LIN {X 0,Y 576.625,Z 290.656,A -85,B 0,C 180,E1 26803.866,E2 26803.866} C_VEL
LIN {X 0,Y 576.086,Z 290.719,A -85,B 0,C 180,E1 26803.314,E2 26803.314} C_VEL
LIN {X 0,Y 576.152,Z 290.716,A -85,B 0,C 180,E1 26800.146,E2 26800.146} C_VEL
LIN {X 0,Y 576.097,Z 290.719,A -85,B 0,C 180,E1 26797.014,E2 26797.014} C_VEL
LIN {X 0,Y 576.121,Z 290.717,A -85,B 0,C 180,E1 26793.733,E2 26793.733} C_VEL
LIN {X 0,Y 576.119,Z 290.718,A -85,B 0,C 180,E1 26790.698,E2 26790.698} C_VEL
LIN {X 0,Y 576.11,Z 290.716,A -85,B 0,C 180,E1 26787.451,E2 26787.451} C_VEL
LIN {X 0,Y 576.157,Z 290.721,A -85,B 0,C 180,E1 26784.306,E2 26784.306} C_VEL
LIN {X 0,Y 576.107,Z 290.717,A -85,B 0,C 180,E1 26781.077,E2 26781.077} C_VEL
LIN {X 0,Y 576.158,Z 290.714,A -85,B 0,C 180,E1 26777.809,E2 26777.809} C_VEL
LIN {X 0,Y 576.125,Z 290.717,A -85,B 0,C 180,E1 26774.638,E2 26774.638} C_VEL
LIN {X 0,Y 576.124,Z 290.716,A -85,B 0,C 180,E1 26771.259,E2 26771.259} C_VEL
LIN {X 0,Y 576.159,Z 290.714,A -85,B 0,C 180,E1 26768.013,E2 26768.013} C_VEL
LIN {X 0,Y 576.122,Z 290.716,A -85,B 0,C 180,E1 26764.817,E2 26764.817} C_VEL
LIN {X 0,Y 576.157,Z 290.709,A -85,B 0,C 180,E1 26761.561,E2 26761.561} C_VEL
LIN {X 0,Y 576.149,Z 290.712,A -85,B 0,C 180,E1 26758.278,E2 26758.278} C_VEL
LIN {X 0,Y 576.195,Z 290.958,A -85,B 0,C 180,E1 26757.573,E2 26757.573} C_VEL
LIN {X 0,Y 578.029,Z 297.635,A -85,B 0,C 180,E1 26756.802,E2 26756.802} C_VEL
LIN {X 0,Y 577.51,Z 328.552,A -85,B 0,C 180,E1 26754.007,E2 26754.007} C_VEL
LIN {X 0,Y 577.497,Z 334.474,A -85,B 0,C 180,E1 26753.515,E2 26753.515} C_VEL
LIN {X 0,Y 578.386,Z 340.749,A -85,B 0,C 180,E1 26753.384,E2 26753.384} C_VEL
LIN {X 0,Y 577.84,Z 542.427,A -85,B 0,C 180,E1 26750.729,E2 26750.729} C_VEL
LIN {X 0,Y 577.686,Z 561.472,A -85,B 0,C 180,E1 26750.287,E2 26750.287} C_VEL
LIN {X 0,Y 577.482,Z 579.605,A -85,B 0,C 180,E1 26749.679,E2 26749.679} C_VEL
LIN {X 0,Y 577.264,Z 597.202,A -85,B 0,C 180,E1 26748.898,E2 26748.898} C_VEL
LIN {X 0,Y 577.039,Z 613.981,A -85,B 0,C 180,E1 26747.959,E2 26747.959} C_VEL
LIN {X 0,Y 576.792,Z 630.391,A -85,B 0,C 180,E1 26746.827,E2 26746.827} C_VEL
LIN {X 0,Y 576.559,Z 645.743,A -85,B 0,C 180,E1 26745.541,E2 26745.541} C_VEL
LIN {X 0,Y 576.356,Z 659.744,A -85,B 0,C 180,E1 26744.128,E2 26744.128} C_VEL
LIN {X 0,Y 576.203,Z 672.121,A -85,B 0,C 180,E1 26742.629,E2 26742.629} C_VEL
LIN {X 0,Y 576.085,Z 683.222,A -85,B 0,C 180,E1 26741.006,E2 26741.006} C_VEL
LIN {X 0,Y 576.006,Z 692.795,A -85,B 0,C 180,E1 26739.29,E2 26739.29} C_VEL
LIN {X 0,Y 575.956,Z 700.403,A -85,B 0,C 180,E1 26737.581,E2 26737.581} C_VEL
LIN {X 0,Y 575.92,Z 706.58,A -85,B 0,C 180,E1 26735.779,E2 26735.779} C_VEL
LIN {X 0,Y 575.92,Z 710.989,A -85,B 0,C 180,E1 26733.982,E2 26733.982} C_VEL
LIN {X 0,Y 575.917,Z 713.852,A -85,B 0,C 180,E1 26732.089,E2 26732.089} C_VEL
LIN {X 0,Y 575.911,Z 714.951,A -85,B 0,C 180,E1 26730.199,E2 26730.199} C_VEL
LIN {X 0,Y 575.913,Z 714.311,A -85,B 0,C 180,E1 26728.309,E2 26728.309} C_VEL
LIN {X 0,Y 575.909,Z 711.917,A -85,B 0,C 180,E1 26726.417,E2 26726.417} C_VEL
LIN {X 0,Y 575.922,Z 707.958,A -85,B 0,C 180,E1 26724.621,E2 26724.621} C_VEL
LIN {X 0,Y 575.945,Z 702.275,A -85,B 0,C 180,E1 26722.82,E2 26722.82} C_VEL
LIN {X 0,Y 575.981,Z 695.171,A -85,B 0,C 180,E1 26721.113,E2 26721.113} C_VEL
LIN {X 0,Y 576.057,Z 686.195,A -85,B 0,C 180,E1 26719.398,E2 26719.398} C_VEL
LIN {X 0,Y 576.164,Z 675.759,A -85,B 0,C 180,E1 26717.777,E2 26717.777} C_VEL
LIN {X 0,Y 576.31,Z 663.875,A -85,B 0,C 180,E1 26716.25,E2 26716.25} C_VEL
LIN {X 0,Y 576.497,Z 650.514,A -85,B 0,C 180,E1 26714.818,E2 26714.818} C_VEL
LIN {X 0,Y 576.72,Z 635.525,A -85,B 0,C 180,E1 26713.482,E2 26713.482} C_VEL
LIN {X 0,Y 576.962,Z 619.334,A -85,B 0,C 180,E1 26712.294,E2 26712.294} C_VEL
LIN {X 0,Y 577.183,Z 602.928,A -85,B 0,C 180,E1 26711.309,E2 26711.309} C_VEL
LIN {X 0,Y 577.431,Z 584.941,A -85,B 0,C 180,E1 26710.448,E2 26710.448} C_VEL
LIN {X 0,Y 577.637,Z 566.861,A -85,B 0,C 180,E1 26709.786,E2 26709.786} C_VEL
LIN {X 0,Y 577.801,Z 548.295,A -85,B 0,C 180,E1 26709.299,E2 26709.299} C_VEL
LIN {X 0,Y 577.907,Z 527.535,A -85,B 0,C 180,E1 26708.962,E2 26708.962} C_VEL
LIN {X 0,Y 578.217,Z 338.32,A -85,B 0,C 180,E1 26706.486,E2 26706.486} C_VEL
LIN {X 0,Y 577.47,Z 334.235,A -85,B 0,C 180,E1 26706.384,E2 26706.384} C_VEL
LIN {X 0,Y 577.872,Z 304.731,A -85,B 0,C 180,E1 26703.764,E2 26703.764} C_VEL
LIN {X 0,Y 577.859,Z 296.714,A -85,B 0,C 180,E1 26703.012,E2 26703.012} C_VEL
LIN {X 0,Y 576.195,Z 290.995,A -85,B 0,C 180,E1 26702.343,E2 26702.343} C_VEL
LIN {X 0,Y 576.146,Z 290.717,A -85,B 0,C 180,E1 26700.7,E2 26700.7} C_VEL
LIN {X 0,Y 576.133,Z 290.719,A -85,B 0,C 180,E1 26697.321,E2 26697.321} C_VEL
LIN {X 0,Y 576.154,Z 290.714,A -85,B 0,C 180,E1 26694.088,E2 26694.088} C_VEL
LIN {X 0,Y 576.124,Z 290.711,A -85,B 0,C 180,E1 26690.875,E2 26690.875} C_VEL
LIN {X 0,Y 576.153,Z 290.716,A -85,B 0,C 180,E1 26687.671,E2 26687.671} C_VEL
LIN {X 0,Y 576.149,Z 290.711,A -85,B 0,C 180,E1 26684.359,E2 26684.359} C_VEL
LIN {X 0,Y 576.119,Z 290.717,A -85,B 0,C 180,E1 26681.129,E2 26681.129} C_VEL
LIN {X 0,Y 576.161,Z 290.716,A -85,B 0,C 180,E1 26677.903,E2 26677.903} C_VEL
LIN {X 0,Y 576.111,Z 290.715,A -85,B 0,C 180,E1 26674.699,E2 26674.699} C_VEL
LIN {X 0,Y 576.145,Z 290.72,A -85,B 0,C 180,E1 26671.491,E2 26671.491} C_VEL
LIN {X 0,Y 576.118,Z 290.715,A -85,B 0,C 180,E1 26668.373,E2 26668.373} C_VEL
LIN {X 0,Y 576.107,Z 290.716,A -85,B 0,C 180,E1 26665.052,E2 26665.052} C_VEL
LIN {X 0,Y 576.151,Z 290.716,A -85,B 0,C 180,E1 26661.908,E2 26661.908} C_VEL
LIN {X 0,Y 576.091,Z 290.717,A -85,B 0,C 180,E1 26658.729,E2 26658.729} C_VEL
LIN {X 0,Y 576.158,Z 290.719,A -85,B 0,C 180,E1 26655.604,E2 26655.604} C_VEL
LIN {X 0,Y 576.085,Z 290.719,A -85,B 0,C 180,E1 26652.53,E2 26652.53} C_VEL
LIN {X 0,Y 576.138,Z 290.717,A -85,B 0,C 180,E1 26649.389,E2 26649.389} C_VEL
LIN {X 0,Y 576.083,Z 290.72,A -85,B 0,C 180,E1 26646.378,E2 26646.378} C_VEL
LIN {X 0,Y 576.113,Z 290.717,A -85,B 0,C 180,E1 26643.184,E2 26643.184} C_VEL
LIN {X 0,Y 576.078,Z 290.721,A -85,B 0,C 180,E1 26640.199,E2 26640.199} C_VEL
LIN {X 0,Y 576.086,Z 290.718,A -85,B 0,C 180,E1 26636.816,E2 26636.816} C_VEL
LIN {X 0,Y 576.111,Z 290.721,A -85,B 0,C 180,E1 26633.823,E2 26633.823} C_VEL
LIN {X 0,Y 576.086,Z 290.719,A -85,B 0,C 180,E1 26630.611,E2 26630.611} C_VEL
LIN {X 0,Y 576.154,Z 290.718,A -85,B 0,C 180,E1 26627.472,E2 26627.472} C_VEL
LIN {X 0,Y 576.089,Z 290.719,A -85,B 0,C 180,E1 26624.291,E2 26624.291} C_VEL
LIN {X 0,Y 576.153,Z 290.716,A -85,B 0,C 180,E1 26621.169,E2 26621.169} C_VEL
LIN {X 0,Y 576.099,Z 290.719,A -85,B 0,C 180,E1 26618.09,E2 26618.09} C_VEL
LIN {X 0,Y 576.131,Z 290.716,A -85,B 0,C 180,E1 26614.838,E2 26614.838} C_VEL
LIN {X 0,Y 576.123,Z 290.718,A -85,B 0,C 180,E1 26611.72,E2 26611.72} C_VEL
LIN {X 0,Y 576.11,Z 290.716,A -85,B 0,C 180,E1 26608.39,E2 26608.39} C_VEL
LIN {X 0,Y 576.16,Z 290.71,A -85,B 0,C 180,E1 26605.166,E2 26605.166} C_VEL
LIN {X 0,Y 576.113,Z 290.716,A -85,B 0,C 180,E1 26601.967,E2 26601.967} C_VEL
LIN {X 0,Y 576.149,Z 290.705,A -85,B 0,C 180,E1 26598.713,E2 26598.713} C_VEL
LIN {X 0,Y 576.145,Z 290.721,A -85,B 0,C 180,E1 26595.484,E2 26595.484} C_VEL
LIN {X 0,Y 576.123,Z 290.716,A -85,B 0,C 180,E1 26592.179,E2 26592.179} C_VEL
LIN {X 0,Y 576.158,Z 290.717,A -85,B 0,C 180,E1 26588.972,E2 26588.972} C_VEL
LIN {X 0,Y 576.132,Z 290.724,A -85,B 0,C 180,E1 26585.669,E2 26585.669} C_VEL
LIN {X 0,Y 576.212,Z 291.106,A -85,B 0,C 180,E1 26585.297,E2 26585.297} C_VEL
LIN {X 0,Y 580.102,Z 300.579,A -85,B 0,C 180,E1 26584.425,E2 26584.425} C_VEL
LIN {X 0,Y 579.434,Z 352.01,A -85,B 0,C 180,E1 26581.407,E2 26581.407} C_VEL
LIN {X 0,Y 579.088,Z 391.09,A -85,B 0,C 180,E1 26579.196,E2 26579.196} C_VEL
LIN {X 0,Y 579.657,Z 397.448,A -85,B 0,C 180,E1 26579.075,E2 26579.075} C_VEL
LIN {X 0,Y 578.923,Z 631.85,A -85,B 0,C 180,E1 26575.903,E2 26575.903} C_VEL
LIN {X 0,Y 578.772,Z 658.475,A -85,B 0,C 180,E1 26575.487,E2 26575.487} C_VEL
LIN {X 0,Y 578.553,Z 678.687,A -85,B 0,C 180,E1 26574.988,E2 26574.988} C_VEL
LIN {X 0,Y 578.317,Z 698.879,A -85,B 0,C 180,E1 26574.297,E2 26574.297} C_VEL
LIN {X 0,Y 578.011,Z 718.11,A -85,B 0,C 180,E1 26573.444,E2 26573.444} C_VEL
LIN {X 0,Y 577.68,Z 736.382,A -85,B 0,C 180,E1 26572.444,E2 26572.444} C_VEL
LIN {X 0,Y 577.339,Z 754.925,A -85,B 0,C 180,E1 26571.22,E2 26571.22} C_VEL
LIN {X 0,Y 577.023,Z 772.23,A -85,B 0,C 180,E1 26569.853,E2 26569.853} C_VEL
LIN {X 0,Y 576.738,Z 788.212,A -85,B 0,C 180,E1 26568.363,E2 26568.363} C_VEL
LIN {X 0,Y 576.505,Z 802.557,A -85,B 0,C 180,E1 26566.793,E2 26566.793} C_VEL
LIN {X 0,Y 576.304,Z 815.862,A -85,B 0,C 180,E1 26565.084,E2 26565.084} C_VEL
LIN {X 0,Y 576.155,Z 828.148,A -85,B 0,C 180,E1 26563.206,E2 26563.206} C_VEL
LIN {X 0,Y 576.041,Z 838.568,A -85,B 0,C 180,E1 26561.277,E2 26561.277} C_VEL
LIN {X 0,Y 575.978,Z 846.875,A -85,B 0,C 180,E1 26559.391,E2 26559.391} C_VEL
LIN {X 0,Y 575.935,Z 853.9,A -85,B 0,C 180,E1 26557.381,E2 26557.381} C_VEL
LIN {X 0,Y 575.916,Z 859.144,A -85,B 0,C 180,E1 26555.379,E2 26555.379} C_VEL
LIN {X 0,Y 575.909,Z 862.738,A -85,B 0,C 180,E1 26553.363,E2 26553.363} C_VEL
LIN {X 0,Y 575.905,Z 864.64,A -85,B 0,C 180,E1 26551.293,E2 26551.293} C_VEL
LIN {X 0,Y 575.904,Z 864.851,A -85,B 0,C 180,E1 26549.304,E2 26549.304} C_VEL
LIN {X 0,Y 575.912,Z 863.392,A -85,B 0,C 180,E1 26547.214,E2 26547.214} C_VEL
LIN {X 0,Y 575.921,Z 860.169,A -85,B 0,C 180,E1 26545.12,E2 26545.12} C_VEL
LIN {X 0,Y 575.935,Z 855.414,A -85,B 0,C 180,E1 26543.12,E2 26543.12} C_VEL
LIN {X 0,Y 575.961,Z 848.851,A -85,B 0,C 180,E1 26541.112,E2 26541.112} C_VEL
LIN {X 0,Y 576.009,Z 840.796,A -85,B 0,C 180,E1 26539.195,E2 26539.195} C_VEL
LIN {X 0,Y 576.104,Z 830.84,A -85,B 0,C 180,E1 26537.267,E2 26537.267} C_VEL
LIN {X 0,Y 576.251,Z 819.393,A -85,B 0,C 180,E1 26535.429,E2 26535.429} C_VEL
LIN {X 0,Y 576.434,Z 806.45,A -85,B 0,C 180,E1 26533.681,E2 26533.681} C_VEL
LIN {X 0,Y 576.677,Z 791.978,A -85,B 0,C 180,E1 26532.024,E2 26532.024} C_VEL
LIN {X 0,Y 576.958,Z 776.494,A -85,B 0,C 180,E1 26530.517,E2 26530.517} C_VEL
LIN {X 0,Y 577.285,Z 759.282,A -85,B 0,C 180,E1 26529.097,E2 26529.097} C_VEL
LIN {X 0,Y 577.625,Z 740.912,A -85,B 0,C 180,E1 26527.831,E2 26527.831} C_VEL
LIN {X 0,Y 577.928,Z 722.295,A -85,B 0,C 180,E1 26526.769,E2 26526.769} C_VEL
LIN {X 0,Y 578.217,Z 703.186,A -85,B 0,C 180,E1 26525.881,E2 26525.881} C_VEL
LIN {X 0,Y 578.509,Z 682.546,A -85,B 0,C 180,E1 26525.132,E2 26525.132} C_VEL
LIN {X 0,Y 578.751,Z 662.256,A -85,B 0,C 180,E1 26524.592,E2 26524.592} C_VEL
LIN {X 0,Y 578.896,Z 641.479,A -85,B 0,C 180,E1 26524.225,E2 26524.225} C_VEL
LIN {X 0,Y 579.633,Z 403.425,A -85,B 0,C 180,E1 26521.007,E2 26521.007} C_VEL
LIN {X 0,Y 579.421,Z 393.381,A -85,B 0,C 180,E1 26520.856,E2 26520.856} C_VEL
LIN {X 0,Y 578.998,Z 389.593,A -85,B 0,C 180,E1 26520.745,E2 26520.745} C_VEL
LIN {X 0,Y 579.691,Z 333.246,A -85,B 0,C 180,E1 26517.504,E2 26517.504} C_VEL
LIN {X 0,Y 580.101,Z 300.579,A -85,B 0,C 180,E1 26515.575,E2 26515.575} C_VEL
LIN {X 0,Y 576.219,Z 291.141,A -85,B 0,C 180,E1 26514.704,E2 26514.704} C_VEL
LIN {X 0,Y 576.132,Z 290.723,A -85,B 0,C 180,E1 26514.311,E2 26514.311} C_VEL
LIN {X 0,Y 576.158,Z 290.717,A -85,B 0,C 180,E1 26511.028,E2 26511.028} C_VEL
LIN {X 0,Y 576.124,Z 290.716,A -85,B 0,C 180,E1 26507.808,E2 26507.808} C_VEL
LIN {X 0,Y 576.144,Z 290.721,A -85,B 0,C 180,E1 26504.501,E2 26504.501} C_VEL
LIN {X 0,Y 576.152,Z 290.704,A -85,B 0,C 180,E1 26501.258,E2 26501.258} C_VEL
LIN {X 0,Y 576.114,Z 290.716,A -85,B 0,C 180,E1 26498.01,E2 26498.01} C_VEL
LIN {X 0,Y 576.16,Z 290.71,A -85,B 0,C 180,E1 26494.816,E2 26494.816} C_VEL
LIN {X 0,Y 576.11,Z 290.716,A -85,B 0,C 180,E1 26491.61,E2 26491.61} C_VEL
LIN {X 0,Y 576.125,Z 290.718,A -85,B 0,C 180,E1 26488.28,E2 26488.28} C_VEL
LIN {X 0,Y 576.132,Z 290.716,A -85,B 0,C 180,E1 26485.162,E2 26485.162} C_VEL
LIN {X 0,Y 576.101,Z 290.719,A -85,B 0,C 180,E1 26481.91,E2 26481.91} C_VEL
LIN {X 0,Y 576.161,Z 290.717,A -85,B 0,C 180,E1 26478.726,E2 26478.726} C_VEL
LIN {X 0,Y 576.092,Z 290.719,A -85,B 0,C 180,E1 26475.587,E2 26475.587} C_VEL
LIN {X 0,Y 576.146,Z 290.721,A -85,B 0,C 180,E1 26472.427,E2 26472.427} C_VEL
LIN {X 0,Y 576.088,Z 290.718,A -85,B 0,C 180,E1 26469.389,E2 26469.389} C_VEL
LIN {X 0,Y 576.117,Z 290.721,A -85,B 0,C 180,E1 26466.177,E2 26466.177} C_VEL
LIN {X 0,Y 576.088,Z 290.718,A -85,B 0,C 180,E1 26463.184,E2 26463.184} C_VEL
LIN {X 0,Y 576.084,Z 290.721,A -85,B 0,C 180,E1 26459.801,E2 26459.801} C_VEL
LIN {X 0,Y 576.107,Z 290.718,A -85,B 0,C 180,E1 26456.816,E2 26456.816} C_VEL
LIN {X 0,Y 576.078,Z 290.72,A -85,B 0,C 180,E1 26453.622,E2 26453.622} C_VEL
LIN {X 0,Y 576.116,Z 290.717,A -85,B 0,C 180,E1 26450.711,E2 26450.711} C_VEL
LIN {X 0,Y 576.084,Z 290.719,A -85,B 0,C 180,E1 26447.572,E2 26447.572} C_VEL
LIN {X 0,Y 576.144,Z 290.717,A -85,B 0,C 180,E1 26444.499,E2 26444.499} C_VEL
LIN {X 0,Y 576.086,Z 290.719,A -85,B 0,C 180,E1 26443.314,E2 26443.314} C_VEL
LIN {X 0,Y 575.12,Z 290.849,A -85,B 0,C 180,E1 26442.548,E2 26442.548} C_VEL
LIN {X 0,Y 568.65,Z 291.651,A -85,B 0,C 180,E1 26440.342,E2 26440.342} C_VEL
LIN {X 0,Y 568.18,Z 291.705,A -85,B 0,C 180,E1 26439.837,E2 26439.837} C_VEL
LIN {X 0,Y 568.172,Z 291.709,A -85,B 0,C 180,E1 26436.784,E2 26436.784} C_VEL
LIN {X 0,Y 568.163,Z 291.707,A -85,B 0,C 180,E1 26433.449,E2 26433.449} C_VEL
LIN {X 0,Y 568.223,Z 291.705,A -85,B 0,C 180,E1 26430.25,E2 26430.25} C_VEL
LIN {X 0,Y 568.163,Z 291.707,A -85,B 0,C 180,E1 26427.058,E2 26427.058} C_VEL
LIN {X 0,Y 568.217,Z 291.704,A -85,B 0,C 180,E1 26423.867,E2 26423.867} C_VEL
LIN {X 0,Y 568.181,Z 291.708,A -85,B 0,C 180,E1 26420.69,E2 26420.69} C_VEL
LIN {X 0,Y 568.182,Z 291.705,A -85,B 0,C 180,E1 26417.351,E2 26417.351} C_VEL
LIN {X 0,Y 568.22,Z 291.697,A -85,B 0,C 180,E1 26414.116,E2 26414.116} C_VEL
LIN {X 0,Y 568.178,Z 291.707,A -85,B 0,C 180,E1 26410.89,E2 26410.89} C_VEL
LIN {X 0,Y 568.217,Z 291.702,A -85,B 0,C 180,E1 26407.631,E2 26407.631} C_VEL
LIN {X 0,Y 568.213,Z 291.7,A -85,B 0,C 180,E1 26404.269,E2 26404.269} C_VEL
LIN {X 0,Y 568.188,Z 291.7,A -85,B 0,C 180,E1 26401.019,E2 26401.019} C_VEL
LIN {X 0,Y 568.24,Z 291.869,A -85,B 0,C 180,E1 26397.992,E2 26397.992} C_VEL
LIN {X 0,Y 570.698,Z 300.422,A -85,B 0,C 180,E1 26396.985,E2 26396.985} C_VEL
LIN {X 0,Y 569.938,Z 334.437,A -85,B 0,C 180,E1 26393.858,E2 26393.858} C_VEL
LIN {X 0,Y 571.042,Z 341.802,A -85,B 0,C 180,E1 26393.69,E2 26393.69} C_VEL
LIN {X 0,Y 570.357,Z 542.461,A -85,B 0,C 180,E1 26391.014,E2 26391.014} C_VEL
LIN {X 0,Y 570.168,Z 561.439,A -85,B 0,C 180,E1 26390.568,E2 26390.568} C_VEL
LIN {X 0,Y 569.912,Z 579.619,A -85,B 0,C 180,E1 26389.951,E2 26389.951} C_VEL
LIN {X 0,Y 569.638,Z 597.212,A -85,B 0,C 180,E1 26389.161,E2 26389.161} C_VEL
LIN {X 0,Y 569.346,Z 613.904,A -85,B 0,C 180,E1 26388.215,E2 26388.215} C_VEL
LIN {X 0,Y 569.043,Z 630.096,A -85,B 0,C 180,E1 26387.087,E2 26387.087} C_VEL
LIN {X 0,Y 568.755,Z 645.194,A -85,B 0,C 180,E1 26385.812,E2 26385.812} C_VEL
LIN {X 0,Y 568.513,Z 658.551,A -85,B 0,C 180,E1 26384.462,E2 26384.462} C_VEL
LIN {X 0,Y 568.303,Z 671.355,A -85,B 0,C 180,E1 26382.911,E2 26382.911} C_VEL
LIN {X 0,Y 568.139,Z 682.59,A -85,B 0,C 180,E1 26381.265,E2 26381.265} C_VEL
LIN {X 0,Y 568.028,Z 692.284,A -85,B 0,C 180,E1 26379.524,E2 26379.524} C_VEL
LIN {X 0,Y 567.964,Z 700.001,A -85,B 0,C 180,E1 26377.79,E2 26377.79} C_VEL
LIN {X 0,Y 567.93,Z 706.281,A -85,B 0,C 180,E1 26375.962,E2 26375.962} C_VEL
LIN {X 0,Y 567.92,Z 710.991,A -85,B 0,C 180,E1 26374.038,E2 26374.038} C_VEL
LIN {X 0,Y 567.917,Z 713.854,A -85,B 0,C 180,E1 26372.119,E2 26372.119} C_VEL
LIN {X 0,Y 567.911,Z 714.951,A -85,B 0,C 180,E1 26370.202,E2 26370.202} C_VEL
LIN {X 0,Y 567.913,Z 714.31,A -85,B 0,C 180,E1 26368.285,E2 26368.285} C_VEL
LIN {X 0,Y 567.911,Z 711.916,A -85,B 0,C 180,E1 26366.366,E2 26366.366} C_VEL
LIN {X 0,Y 567.926,Z 707.956,A -85,B 0,C 180,E1 26364.545,E2 26364.545} C_VEL
LIN {X 0,Y 567.952,Z 702.272,A -85,B 0,C 180,E1 26362.718,E2 26362.718} C_VEL
LIN {X 0,Y 568.01,Z 694.957,A -85,B 0,C 180,E1 26360.94,E2 26360.94} C_VEL
LIN {X 0,Y 568.097,Z 686.193,A -85,B 0,C 180,E1 26359.248,E2 26359.248} C_VEL
LIN {X 0,Y 568.244,Z 675.52,A -85,B 0,C 180,E1 26357.57,E2 26357.57} C_VEL
LIN {X 0,Y 568.423,Z 663.87,A -85,B 0,C 180,E1 26356.056,E2 26356.056} C_VEL
LIN {X 0,Y 568.659,Z 650.506,A -85,B 0,C 180,E1 26354.604,E2 26354.604} C_VEL
LIN {X 0,Y 568.942,Z 635.518,A -85,B 0,C 180,E1 26353.25,E2 26353.25} C_VEL
LIN {X 0,Y 569.246,Z 619.329,A -85,B 0,C 180,E1 26352.046,E2 26352.046} C_VEL
LIN {X 0,Y 569.532,Z 602.921,A -85,B 0,C 180,E1 26351.048,E2 26351.048} C_VEL
LIN {X 0,Y 569.835,Z 585.631,A -85,B 0,C 180,E1 26350.206,E2 26350.206} C_VEL
LIN {X 0,Y 570.095,Z 567.459,A -85,B 0,C 180,E1 26349.526,E2 26349.526} C_VEL
LIN {X 0,Y 570.302,Z 548.912,A -85,B 0,C 180,E1 26349.028,E2 26349.028} C_VEL
LIN {X 0,Y 570.433,Z 528.629,A -85,B 0,C 180,E1 26348.688,E2 26348.688} C_VEL
LIN {X 0,Y 570.885,Z 339.627,A -85,B 0,C 180,E1 26346.184,E2 26346.184} C_VEL
LIN {X 0,Y 569.914,Z 334.093,A -85,B 0,C 180,E1 26346.032,E2 26346.032} C_VEL
LIN {X 0,Y 570.703,Z 300.17,A -85,B 0,C 180,E1 26342.903,E2 26342.903} C_VEL
LIN {X 0,Y 568.242,Z 291.898,A -85,B 0,C 180,E1 26341.922,E2 26341.922} C_VEL
LIN {X 0,Y 568.211,Z 291.697,A -85,B 0,C 180,E1 26338.611,E2 26338.611} C_VEL
LIN {X 0,Y 568.191,Z 291.705,A -85,B 0,C 180,E1 26335.265,E2 26335.265} C_VEL
LIN {X 0,Y 568.218,Z 291.702,A -85,B 0,C 180,E1 26331.986,E2 26331.986} C_VEL
LIN {X 0,Y 568.19,Z 291.704,A -85,B 0,C 180,E1 26328.709,E2 26328.709} C_VEL
LIN {X 0,Y 568.191,Z 291.705,A -85,B 0,C 180,E1 26325.311,E2 26325.311} C_VEL
LIN {X 0,Y 568.221,Z 291.704,A -85,B 0,C 180,E1 26322.052,E2 26322.052} C_VEL
LIN {X 0,Y 568.175,Z 291.705,A -85,B 0,C 180,E1 26318.78,E2 26318.78} C_VEL
LIN {X 0,Y 568.206,Z 291.708,A -85,B 0,C 180,E1 26315.5,E2 26315.5} C_VEL
LIN {X 0,Y 568.188,Z 291.704,A -85,B 0,C 180,E1 26312.341,E2 26312.341} C_VEL
LIN {X 0,Y 568.171,Z 291.706,A -85,B 0,C 180,E1 26309.059,E2 26309.059} C_VEL
LIN {X 0,Y 568.219,Z 291.705,A -85,B 0,C 180,E1 26305.874,E2 26305.874} C_VEL
LIN {X 0,Y 568.159,Z 291.707,A -85,B 0,C 180,E1 26302.669,E2 26302.669} C_VEL
LIN {X 0,Y 568.199,Z 291.707,A -85,B 0,C 180,E1 26299.426,E2 26299.426} C_VEL
LIN {X 0,Y 568.16,Z 291.707,A -85,B 0,C 180,E1 26296.354,E2 26296.354} C_VEL
LIN {X 0,Y 568.161,Z 291.708,A -85,B 0,C 180,E1 26293.018,E2 26293.018} C_VEL
LIN {X 0,Y 568.173,Z 291.707,A -85,B 0,C 180,E1 26290.033,E2 26290.033} C_VEL
LIN {X 0,Y 568.144,Z 291.709,A -85,B 0,C 180,E1 26286.772,E2 26286.772} C_VEL
LIN {X 0,Y 568.206,Z 291.708,A -85,B 0,C 180,E1 26283.632,E2 26283.632} C_VEL
LIN {X 0,Y 568.134,Z 291.71,A -85,B 0,C 180,E1 26280.504,E2 26280.504} C_VEL
LIN {X 0,Y 568.204,Z 291.705,A -85,B 0,C 180,E1 26277.378,E2 26277.378} C_VEL
LIN {X 0,Y 568.143,Z 291.709,A -85,B 0,C 180,E1 26274.243,E2 26274.243} C_VEL
LIN {X 0,Y 568.173,Z 291.707,A -85,B 0,C 180,E1 26270.989,E2 26270.989} C_VEL
LIN {X 0,Y 568.158,Z 291.709,A -85,B 0,C 180,E1 26268.015,E2 26268.015} C_VEL
LIN {X 0,Y 568.159,Z 291.708,A -85,B 0,C 180,E1 26264.656,E2 26264.656} C_VEL
LIN {X 0,Y 568.193,Z 291.708,A -85,B 0,C 180,E1 26261.64,E2 26261.64} C_VEL
LIN {X 0,Y 568.158,Z 291.707,A -85,B 0,C 180,E1 26258.42,E2 26258.42} C_VEL
LIN {X 0,Y 568.224,Z 291.706,A -85,B 0,C 180,E1 26255.222,E2 26255.222} C_VEL
LIN {X 0,Y 568.164,Z 291.706,A -85,B 0,C 180,E1 26252.055,E2 26252.055} C_VEL
LIN {X 0,Y 568.198,Z 291.703,A -85,B 0,C 180,E1 26248.781,E2 26248.781} C_VEL
LIN {X 0,Y 568.194,Z 291.709,A -85,B 0,C 180,E1 26245.607,E2 26245.607} C_VEL
LIN {X 0,Y 568.178,Z 291.703,A -85,B 0,C 180,E1 26242.361,E2 26242.361} C_VEL
LIN {X 0,Y 568.221,Z 291.697,A -85,B 0,C 180,E1 26239.167,E2 26239.167} C_VEL
LIN {X 0,Y 568.181,Z 291.708,A -85,B 0,C 180,E1 26235.886,E2 26235.886} C_VEL
LIN {X 0,Y 568.213,Z 291.703,A -85,B 0,C 180,E1 26232.644,E2 26232.644} C_VEL
LIN {X 0,Y 568.219,Z 291.7,A -85,B 0,C 180,E1 26229.264,E2 26229.264} C_VEL
LIN {X 0,Y 568.189,Z 291.725,A -85,B 0,C 180,E1 26225.956,E2 26225.956} C_VEL
LIN {X 0,Y 568.299,Z 292.358,A -85,B 0,C 180,E1 26225.739,E2 26225.739} C_VEL
LIN {X 0,Y 573.205,Z 304.206,A -85,B 0,C 180,E1 26224.675,E2 26224.675} C_VEL
LIN {X 0,Y 572.309,Z 356.956,A -85,B 0,C 180,E1 26221.549,E2 26221.549} C_VEL
LIN {X 0,Y 571.927,Z 391.105,A -85,B 0,C 180,E1 26219.597,E2 26219.597} C_VEL
LIN {X 0,Y 572.661,Z 398.211,A -85,B 0,C 180,E1 26219.454,E2 26219.454} C_VEL
LIN {X 0,Y 571.722,Z 632.806,A -85,B 0,C 180,E1 26216.241,E2 26216.241} C_VEL
LIN {X 0,Y 571.532,Z 658.962,A -85,B 0,C 180,E1 26215.823,E2 26215.823} C_VEL
LIN {X 0,Y 571.252,Z 679.552,A -85,B 0,C 180,E1 26215.302,E2 26215.302} C_VEL
LIN {X 0,Y 570.968,Z 698.877,A -85,B 0,C 180,E1 26214.63,E2 26214.63} C_VEL
LIN {X 0,Y 570.579,Z 718.114,A -85,B 0,C 180,E1 26213.768,E2 26213.768} C_VEL
LIN {X 0,Y 570.153,Z 737.04,A -85,B 0,C 180,E1 26212.717,E2 26212.717} C_VEL
LIN {X 0,Y 569.744,Z 754.928,A -85,B 0,C 180,E1 26211.516,E2 26211.516} C_VEL
LIN {X 0,Y 569.343,Z 772.232,A -85,B 0,C 180,E1 26210.133,E2 26210.133} C_VEL
LIN {X 0,Y 568.969,Z 788.436,A -85,B 0,C 180,E1 26208.599,E2 26208.599} C_VEL
LIN {X 0,Y 568.661,Z 803.058,A -85,B 0,C 180,E1 26206.97,E2 26206.97} C_VEL
LIN {X 0,Y 568.418,Z 815.863,A -85,B 0,C 180,E1 26205.298,E2 26205.298} C_VEL
LIN {X 0,Y 568.225,Z 827.928,A -85,B 0,C 180,E1 26203.43,E2 26203.43} C_VEL
LIN {X 0,Y 568.078,Z 837.883,A -85,B 0,C 180,E1 26201.575,E2 26201.575} C_VEL
LIN {X 0,Y 567.992,Z 846.469,A -85,B 0,C 180,E1 26199.627,E2 26199.627} C_VEL
LIN {X 0,Y 567.947,Z 853.597,A -85,B 0,C 180,E1 26197.587,E2 26197.587} C_VEL
LIN {X 0,Y 567.925,Z 858.73,A -85,B 0,C 180,E1 26195.658,E2 26195.658} C_VEL
LIN {X 0,Y 567.909,Z 862.558,A -85,B 0,C 180,E1 26193.533,E2 26193.533} C_VEL
LIN {X 0,Y 567.902,Z 864.507,A -85,B 0,C 180,E1 26191.513,E2 26191.513} C_VEL
LIN {X 0,Y 567.9,Z 864.896,A -85,B 0,C 180,E1 26189.496,E2 26189.496} C_VEL
LIN {X 0,Y 567.901,Z 863.728,A -85,B 0,C 180,E1 26187.477,E2 26187.477} C_VEL
LIN {X 0,Y 567.907,Z 860.972,A -85,B 0,C 180,E1 26185.456,E2 26185.456} C_VEL
LIN {X 0,Y 567.926,Z 856.483,A -85,B 0,C 180,E1 26183.429,E2 26183.429} C_VEL
LIN {X 0,Y 567.965,Z 850.267,A -85,B 0,C 180,E1 26181.394,E2 26181.394} C_VEL
LIN {X 0,Y 568.03,Z 842.181,A -85,B 0,C 180,E1 26179.349,E2 26179.349} C_VEL
LIN {X 0,Y 568.145,Z 832.569,A -85,B 0,C 180,E1 26177.396,E2 26177.396} C_VEL
LIN {X 0,Y 568.32,Z 821.497,A -85,B 0,C 180,E1 26175.533,E2 26175.533} C_VEL
LIN {X 0,Y 568.551,Z 808.943,A -85,B 0,C 180,E1 26173.763,E2 26173.763} C_VEL
LIN {X 0,Y 568.837,Z 794.891,A -85,B 0,C 180,E1 26172.086,E2 26172.086} C_VEL
LIN {X 0,Y 569.168,Z 779.848,A -85,B 0,C 180,E1 26170.556,E2 26170.556} C_VEL
LIN {X 0,Y 569.55,Z 763.302,A -85,B 0,C 180,E1 26169.123,E2 26169.123} C_VEL
LIN {X 0,Y 569.976,Z 744.963,A -85,B 0,C 180,E1 26167.789,E2 26167.789} C_VEL
LIN {X 0,Y 570.378,Z 726.292,A -85,B 0,C 180,E1 26166.662,E2 26166.662} C_VEL
LIN {X 0,Y 570.785,Z 707.828,A -85,B 0,C 180,E1 26165.747,E2 26165.747} C_VEL
LIN {X 0,Y 571.158,Z 687.897,A -85,B 0,C 180,E1 26164.964,E2 26164.964} C_VEL
LIN {X 0,Y 571.425,Z 667.643,A -85,B 0,C 180,E1 26164.371,E2 26164.371} C_VEL
LIN {X 0,Y 571.645,Z 647.244,A -85,B 0,C 180,E1 26163.965,E2 26163.965} C_VEL
LIN {X 0,Y 572.627,Z 405.206,A -85,B 0,C 180,E1 26160.643,E2 26160.643} C_VEL
LIN {X 0,Y 572.429,Z 394.559,A -85,B 0,C 180,E1 26160.481,E2 26160.481} C_VEL
LIN {X 0,Y 571.833,Z 389.593,A -85,B 0,C 180,E1 26160.342,E2 26160.342} C_VEL
LIN {X 0,Y 572.729,Z 332.228,A -85,B 0,C 180,E1 26156.998,E2 26156.998} C_VEL
LIN {X 0,Y 573.013,Z 303.541,A -85,B 0,C 180,E1 26155.271,E2 26155.271} C_VEL
LIN {X 0,Y 568.253,Z 292.129,A -85,B 0,C 180,E1 26154.229,E2 26154.229} C_VEL
LIN {X 0,Y 568.189,Z 291.704,A -85,B 0,C 180,E1 26153.873,E2 26153.873} C_VEL
LIN {X 0,Y 568.209,Z 291.699,A -85,B 0,C 180,E1 26150.564,E2 26150.564} C_VEL
LIN {X 0,Y 568.219,Z 291.704,A -85,B 0,C 180,E1 26147.203,E2 26147.203} C_VEL
LIN {X 0,Y 568.179,Z 291.707,A -85,B 0,C 180,E1 26143.969,E2 26143.969} C_VEL
LIN {X 0,Y 568.221,Z 291.7,A -85,B 0,C 180,E1 26140.679,E2 26140.679} C_VEL
LIN {X 0,Y 568.187,Z 291.702,A -85,B 0,C 180,E1 26137.475,E2 26137.475} C_VEL
LIN {X 0,Y 568.178,Z 291.708,A -85,B 0,C 180,E1 26134.15,E2 26134.15} C_VEL
LIN {X 0,Y 568.222,Z 291.703,A -85,B 0,C 180,E1 26130.918,E2 26130.918} C_VEL
LIN {X 0,Y 568.165,Z 291.705,A -85,B 0,C 180,E1 26127.683,E2 26127.683} C_VEL
LIN {X 0,Y 568.202,Z 291.708,A -85,B 0,C 180,E1 26124.426,E2 26124.426} C_VEL
LIN {X 0,Y 568.17,Z 291.706,A -85,B 0,C 180,E1 26121.363,E2 26121.363} C_VEL
LIN {X 0,Y 568.166,Z 291.707,A -85,B 0,C 180,E1 26118.042,E2 26118.042} C_VEL
LIN {X 0,Y 568.192,Z 291.706,A -85,B 0,C 180,E1 26114.971,E2 26114.971} C_VEL
LIN {X 0,Y 568.15,Z 291.709,A -85,B 0,C 180,E1 26111.779,E2 26111.779} C_VEL
LIN {X 0,Y 568.216,Z 291.705,A -85,B 0,C 180,E1 26108.602,E2 26108.602} C_VEL
LIN {X 0,Y 568.143,Z 291.709,A -85,B 0,C 180,E1 26105.453,E2 26105.453} C_VEL
LIN {X 0,Y 568.183,Z 291.708,A -85,B 0,C 180,E1 26102.219,E2 26102.219} C_VEL
LIN {X 0,Y 568.139,Z 291.71,A -85,B 0,C 180,E1 26099.294,E2 26099.294} C_VEL
LIN {X 0,Y 568.169,Z 291.709,A -85,B 0,C 180,E1 26096.064,E2 26096.064} C_VEL
LIN {X 0,Y 568.15,Z 291.71,A -85,B 0,C 180,E1 26093.025,E2 26093.025} C_VEL
LIN {X 0,Y 568.148,Z 291.709,A -85,B 0,C 180,E1 26089.651,E2 26089.651} C_VEL
LIN {X 0,Y 568.197,Z 291.709,A -85,B 0,C 180,E1 26086.568,E2 26086.568} C_VEL
LIN {X 0,Y 568.149,Z 291.708,A -85,B 0,C 180,E1 26083.435,E2 26083.435} C_VEL
LIN {X 0,Y 568.219,Z 291.704,A -85,B 0,C 180,E1 26080.254,E2 26080.254} C_VEL
LIN {X 0,Y 568.18,Z 291.705,A -85,B 0,C 180,E1 26079.837,E2 26079.837} C_VEL
LIN {X 0,Y 567.152,Z 291.832,A -85,B 0,C 180,E1 26079.061,E2 26079.061} C_VEL
LIN {X 0,Y 560.801,Z 292.636,A -85,B 0,C 180,E1 26076.88,E2 26076.88} C_VEL
LIN {X 0,Y 560.282,Z 292.693,A -85,B 0,C 180,E1 26076.313,E2 26076.313} C_VEL
LIN {X 0,Y 560.219,Z 292.697,A -85,B 0,C 180,E1 26073.157,E2 26073.157} C_VEL
LIN {X 0,Y 560.271,Z 292.693,A -85,B 0,C 180,E1 26069.902,E2 26069.902} C_VEL
LIN {X 0,Y 560.236,Z 292.697,A -85,B 0,C 180,E1 26066.776,E2 26066.776} C_VEL
LIN {X 0,Y 560.238,Z 292.694,A -85,B 0,C 180,E1 26063.409,E2 26063.409} C_VEL
LIN {X 0,Y 560.286,Z 292.696,A -85,B 0,C 180,E1 26060.159,E2 26060.159} C_VEL
LIN {X 0,Y 560.236,Z 292.696,A -85,B 0,C 180,E1 26056.879,E2 26056.879} C_VEL
LIN {X 0,Y 560.263,Z 292.684,A -85,B 0,C 180,E1 26053.539,E2 26053.539} C_VEL
LIN {X 0,Y 560.279,Z 292.694,A -85,B 0,C 180,E1 26050.199,E2 26050.199} C_VEL
LIN {X 0,Y 560.243,Z 292.694,A -85,B 0,C 180,E1 26046.913,E2 26046.913} C_VEL
LIN {X 0,Y 560.28,Z 292.691,A -85,B 0,C 180,E1 26043.587,E2 26043.587} C_VEL
LIN {X 0,Y 560.279,Z 292.687,A -85,B 0,C 180,E1 26040.214,E2 26040.214} C_VEL
LIN {X 0,Y 560.305,Z 292.964,A -85,B 0,C 180,E1 26038.387,E2 26038.387} C_VEL
LIN {X 0,Y 563.388,Z 303.018,A -85,B 0,C 180,E1 26037.192,E2 26037.192} C_VEL
LIN {X 0,Y 562.6,Z 334.852,A -85,B 0,C 180,E1 26034.238,E2 26034.238} C_VEL
LIN {X 0,Y 563.916,Z 343.007,A -85,B 0,C 180,E1 26034.045,E2 26034.045} C_VEL
LIN {X 0,Y 562.881,Z 542.819,A -85,B 0,C 180,E1 26031.3,E2 26031.3} C_VEL
LIN {X 0,Y 562.657,Z 561.678,A -85,B 0,C 180,E1 26030.848,E2 26030.848} C_VEL
LIN {X 0,Y 562.355,Z 579.633,A -85,B 0,C 180,E1 26030.231,E2 26030.231} C_VEL
LIN {X 0,Y 562.024,Z 597.222,A -85,B 0,C 180,E1 26029.431,E2 26029.431} C_VEL
LIN {X 0,Y 561.663,Z 613.911,A -85,B 0,C 180,E1 26028.473,E2 26028.473} C_VEL
LIN {X 0,Y 561.306,Z 629.734,A -85,B 0,C 180,E1 26027.359,E2 26027.359} C_VEL
LIN {X 0,Y 560.965,Z 644.403,A -85,B 0,C 180,E1 26026.114,E2 26026.114} C_VEL
LIN {X 0,Y 560.675,Z 657.631,A -85,B 0,C 180,E1 26024.774,E2 26024.774} C_VEL
LIN {X 0,Y 560.424,Z 669.814,A -85,B 0,C 180,E1 26023.306,E2 26023.306} C_VEL
LIN {X 0,Y 560.219,Z 681.321,A -85,B 0,C 180,E1 26021.635,E2 26021.635} C_VEL
LIN {X 0,Y 560.081,Z 690.74,A -85,B 0,C 180,E1 26019.972,E2 26019.972} C_VEL
LIN {X 0,Y 559.997,Z 698.789,A -85,B 0,C 180,E1 26018.212,E2 26018.212} C_VEL
LIN {X 0,Y 559.939,Z 705.374,A -85,B 0,C 180,E1 26016.356,E2 26016.356} C_VEL
LIN {X 0,Y 559.921,Z 710.168,A -85,B 0,C 180,E1 26014.506,E2 26014.506} C_VEL
LIN {X 0,Y 559.907,Z 713.29,A -85,B 0,C 180,E1 26012.661,E2 26012.661} C_VEL
LIN {X 0,Y 559.915,Z 714.838,A -85,B 0,C 180,E1 26010.716,E2 26010.716} C_VEL
LIN {X 0,Y 559.909,Z 714.647,A -85,B 0,C 180,E1 26008.772,E2 26008.772} C_VEL
LIN {X 0,Y 559.914,Z 712.708,A -85,B 0,C 180,E1 26006.827,E2 26006.827} C_VEL
LIN {X 0,Y 559.923,Z 709.223,A -85,B 0,C 180,E1 26004.98,E2 26004.98} C_VEL
LIN {X 0,Y 559.952,Z 704.018,A -85,B 0,C 180,E1 26003.124,E2 26003.124} C_VEL
LIN {X 0,Y 560.005,Z 697.005,A -85,B 0,C 180,E1 26001.271,E2 26001.271} C_VEL
LIN {X 0,Y 560.112,Z 688.488,A -85,B 0,C 180,E1 25999.509,E2 25999.509} C_VEL
LIN {X 0,Y 560.259,Z 678.56,A -85,B 0,C 180,E1 25997.844,E2 25997.844} C_VEL
LIN {X 0,Y 560.47,Z 667.253,A -85,B 0,C 180,E1 25996.275,E2 25996.275} C_VEL
LIN {X 0,Y 560.738,Z 654.562,A -85,B 0,C 180,E1 25994.805,E2 25994.805} C_VEL
LIN {X 0,Y 561.057,Z 640.393,A -85,B 0,C 180,E1 25993.434,E2 25993.434} C_VEL
LIN {X 0,Y 561.423,Z 624.546,A -85,B 0,C 180,E1 25992.163,E2 25992.163} C_VEL
LIN {X 0,Y 561.79,Z 607.513,A -85,B 0,C 180,E1 25991.047,E2 25991.047} C_VEL
LIN {X 0,Y 562.163,Z 590.281,A -85,B 0,C 180,E1 25990.141,E2 25990.141} C_VEL
LIN {X 0,Y 562.487,Z 571.965,A -85,B 0,C 180,E1 25989.394,E2 25989.394} C_VEL
LIN {X 0,Y 562.753,Z 553.456,A -85,B 0,C 180,E1 25988.842,E2 25988.842} C_VEL
LIN {X 0,Y 562.941,Z 534.654,A -85,B 0,C 180,E1 25988.477,E2 25988.477} C_VEL
LIN {X 0,Y 563.774,Z 340.944,A -85,B 0,C 180,E1 25985.83,E2 25985.83} C_VEL
LIN {X 0,Y 562.571,Z 334.474,A -85,B 0,C 180,E1 25985.649,E2 25985.649} C_VEL
LIN {X 0,Y 563.375,Z 302.788,A -85,B 0,C 180,E1 25982.693,E2 25982.693} C_VEL
LIN {X 0,Y 560.303,Z 292.942,A -85,B 0,C 180,E1 25981.517,E2 25981.517} C_VEL
LIN {X 0,Y 560.278,Z 292.686,A -85,B 0,C 180,E1 25978.348,E2 25978.348} C_VEL
LIN {X 0,Y 560.25,Z 292.692,A -85,B 0,C 180,E1 25975.05,E2 25975.05} C_VEL
LIN {X 0,Y 560.277,Z 292.687,A -85,B 0,C 180,E1 25971.74,E2 25971.74} C_VEL
LIN {X 0,Y 560.277,Z 292.691,A -85,B 0,C 180,E1 25968.395,E2 25968.395} C_VEL
LIN {X 0,Y 560.243,Z 292.692,A -85,B 0,C 180,E1 25965.115,E2 25965.115} C_VEL
LIN {X 0,Y 560.283,Z 292.696,A -85,B 0,C 180,E1 25961.869,E2 25961.869} C_VEL
LIN {X 0,Y 560.245,Z 292.693,A -85,B 0,C 180,E1 25958.587,E2 25958.587} C_VEL
LIN {X 0,Y 560.241,Z 292.695,A -85,B 0,C 180,E1 25955.178,E2 25955.178} C_VEL
LIN {X 0,Y 560.285,Z 292.693,A -85,B 0,C 180,E1 25951.886,E2 25951.886} C_VEL
LIN {X 0,Y 560.226,Z 292.694,A -85,B 0,C 180,E1 25948.692,E2 25948.692} C_VEL
LIN {X 0,Y 560.263,Z 292.693,A -85,B 0,C 180,E1 25945.446,E2 25945.446} C_VEL
LIN {X 0,Y 560.233,Z 292.695,A -85,B 0,C 180,E1 25942.343,E2 25942.343} C_VEL
LIN {X 0,Y 560.219,Z 292.695,A -85,B 0,C 180,E1 25938.933,E2 25938.933} C_VEL
LIN {X 0,Y 560.28,Z 292.696,A -85,B 0,C 180,E1 25935.739,E2 25935.739} C_VEL
LIN {X 0,Y 560.208,Z 292.697,A -85,B 0,C 180,E1 25932.577,E2 25932.577} C_VEL
LIN {X 0,Y 560.254,Z 292.692,A -85,B 0,C 180,E1 25929.347,E2 25929.347} C_VEL
LIN {X 0,Y 560.206,Z 292.698,A -85,B 0,C 180,E1 25926.353,E2 25926.353} C_VEL
LIN {X 0,Y 560.223,Z 292.694,A -85,B 0,C 180,E1 25923.069,E2 25923.069} C_VEL
LIN {X 0,Y 560.208,Z 292.699,A -85,B 0,C 180,E1 25920.102,E2 25920.102} C_VEL
LIN {X 0,Y 560.203,Z 292.695,A -85,B 0,C 180,E1 25916.726,E2 25916.726} C_VEL
LIN {X 0,Y 560.269,Z 292.699,A -85,B 0,C 180,E1 25913.545,E2 25913.545} C_VEL
LIN {X 0,Y 560.205,Z 292.697,A -85,B 0,C 180,E1 25910.342,E2 25910.342} C_VEL
LIN {X 0,Y 560.256,Z 292.691,A -85,B 0,C 180,E1 25907.11,E2 25907.11} C_VEL
LIN {X 0,Y 560.219,Z 292.698,A -85,B 0,C 180,E1 25904.047,E2 25904.047} C_VEL
LIN {X 0,Y 560.225,Z 292.695,A -85,B 0,C 180,E1 25900.612,E2 25900.612} C_VEL
LIN {X 0,Y 560.275,Z 292.695,A -85,B 0,C 180,E1 25897.438,E2 25897.438} C_VEL
LIN {X 0,Y 560.223,Z 292.696,A -85,B 0,C 180,E1 25894.184,E2 25894.184} C_VEL
LIN {X 0,Y 560.274,Z 292.693,A -85,B 0,C 180,E1 25890.961,E2 25890.961} C_VEL
LIN {X 0,Y 560.243,Z 292.696,A -85,B 0,C 180,E1 25887.75,E2 25887.75} C_VEL
LIN {X 0,Y 560.238,Z 292.683,A -85,B 0,C 180,E1 25884.422,E2 25884.422} C_VEL
LIN {X 0,Y 560.283,Z 292.697,A -85,B 0,C 180,E1 25881.217,E2 25881.217} C_VEL
LIN {X 0,Y 560.238,Z 292.684,A -85,B 0,C 180,E1 25877.937,E2 25877.937} C_VEL
LIN {X 0,Y 560.268,Z 292.687,A -85,B 0,C 180,E1 25874.598,E2 25874.598} C_VEL
LIN {X 0,Y 560.28,Z 292.695,A -85,B 0,C 180,E1 25871.297,E2 25871.297} C_VEL
LIN {X 0,Y 560.247,Z 292.699,A -85,B 0,C 180,E1 25868.002,E2 25868.002} C_VEL
LIN {X 0,Y 560.282,Z 292.88,A -85,B 0,C 180,E1 25866.262,E2 25866.262} C_VEL
LIN {X 0,Y 560.934,Z 295.081,A -85,B 0,C 180,E1 25866.03,E2 25866.03} C_VEL
LIN {X 0,Y 566.263,Z 307.722,A -85,B 0,C 180,E1 25864.935,E2 25864.935} C_VEL
LIN {X 0,Y 565.204,Z 360.911,A -85,B 0,C 180,E1 25861.754,E2 25861.754} C_VEL
LIN {X 0,Y 564.776,Z 391.023,A -85,B 0,C 180,E1 25860.011,E2 25860.011} C_VEL
LIN {X 0,Y 565.688,Z 399.229,A -85,B 0,C 180,E1 25859.839,E2 25859.839} C_VEL
LIN {X 0,Y 564.542,Z 633.955,A -85,B 0,C 180,E1 25856.585,E2 25856.585} C_VEL
LIN {X 0,Y 564.314,Z 659.286,A -85,B 0,C 180,E1 25856.171,E2 25856.171} C_VEL
LIN {X 0,Y 563.973,Z 680.201,A -85,B 0,C 180,E1 25855.631,E2 25855.631} C_VEL
LIN {X 0,Y 563.598,Z 700.159,A -85,B 0,C 180,E1 25854.918,E2 25854.918} C_VEL
LIN {X 0,Y 563.149,Z 719.236,A -85,B 0,C 180,E1 25854.045,E2 25854.045} C_VEL
LIN {X 0,Y 562.629,Z 738.229,A -85,B 0,C 180,E1 25852.964,E2 25852.964} C_VEL
LIN {X 0,Y 562.143,Z 755.657,A -85,B 0,C 180,E1 25851.767,E2 25851.767} C_VEL
LIN {X 0,Y 561.656,Z 772.838,A -85,B 0,C 180,E1 25850.366,E2 25850.366} C_VEL
LIN {X 0,Y 561.186,Z 789.434,A -85,B 0,C 180,E1 25848.76,E2 25848.76} C_VEL
LIN {X 0,Y 560.814,Z 803.908,A -85,B 0,C 180,E1 25847.107,E2 25847.107} C_VEL
LIN {X 0,Y 560.519,Z 816.571,A -85,B 0,C 180,E1 25845.413,E2 25845.413} C_VEL
LIN {X 0,Y 560.286,Z 828.533,A -85,B 0,C 180,E1 25843.519,E2 25843.519} C_VEL
LIN {X 0,Y 560.111,Z 838.911,A -85,B 0,C 180,E1 25841.533,E2 25841.533} C_VEL
LIN {X 0,Y 560.008,Z 847.28,A -85,B 0,C 180,E1 25839.558,E2 25839.558} C_VEL
LIN {X 0,Y 559.953,Z 853.9,A -85,B 0,C 180,E1 25837.593,E2 25837.593} C_VEL
LIN {X 0,Y 559.922,Z 859.143,A -85,B 0,C 180,E1 25835.533,E2 25835.533} C_VEL
LIN {X 0,Y 559.909,Z 862.71,A -85,B 0,C 180,E1 25833.481,E2 25833.481} C_VEL
LIN {X 0,Y 559.904,Z 864.64,A -85,B 0,C 180,E1 25831.33,E2 25831.33} C_VEL
LIN {X 0,Y 559.905,Z 864.851,A -85,B 0,C 180,E1 25829.284,E2 25829.284} C_VEL
LIN {X 0,Y 559.914,Z 863.393,A -85,B 0,C 180,E1 25827.134,E2 25827.134} C_VEL
LIN {X 0,Y 559.924,Z 860.17,A -85,B 0,C 180,E1 25824.98,E2 25824.98} C_VEL
LIN {X 0,Y 559.947,Z 855.415,A -85,B 0,C 180,E1 25822.923,E2 25822.923} C_VEL
LIN {X 0,Y 559.995,Z 848.852,A -85,B 0,C 180,E1 25820.857,E2 25820.857} C_VEL
LIN {X 0,Y 560.079,Z 840.797,A -85,B 0,C 180,E1 25818.884,E2 25818.884} C_VEL
LIN {X 0,Y 560.235,Z 830.842,A -85,B 0,C 180,E1 25816.9,E2 25816.9} C_VEL
LIN {X 0,Y 560.454,Z 819.394,A -85,B 0,C 180,E1 25815.009,E2 25815.009} C_VEL
LIN {X 0,Y 560.746,Z 806.448,A -85,B 0,C 180,E1 25813.211,E2 25813.211} C_VEL
LIN {X 0,Y 561.103,Z 792.705,A -85,B 0,C 180,E1 25811.585,E2 25811.585} C_VEL
LIN {X 0,Y 561.533,Z 777.056,A -85,B 0,C 180,E1 25810.01,E2 25810.01} C_VEL
LIN {X 0,Y 562.026,Z 759.961,A -85,B 0,C 180,E1 25808.557,E2 25808.557} C_VEL
LIN {X 0,Y 562.532,Z 742.205,A -85,B 0,C 180,E1 25807.291,E2 25807.291} C_VEL
LIN {X 0,Y 562.996,Z 724.297,A -85,B 0,C 180,E1 25806.226,E2 25806.226} C_VEL
LIN {X 0,Y 563.466,Z 704.736,A -85,B 0,C 180,E1 25805.275,E2 25805.275} C_VEL
LIN {X 0,Y 563.906,Z 684.562,A -85,B 0,C 180,E1 25804.508,E2 25804.508} C_VEL
LIN {X 0,Y 564.273,Z 664.469,A -85,B 0,C 180,E1 25803.939,E2 25803.939} C_VEL
LIN {X 0,Y 564.493,Z 643.382,A -85,B 0,C 180,E1 25803.546,E2 25803.546} C_VEL
LIN {X 0,Y 565.655,Z 405.079,A -85,B 0,C 180,E1 25800.243,E2 25800.243} C_VEL
LIN {X 0,Y 565.443,Z 395.593,A -85,B 0,C 180,E1 25800.094,E2 25800.094} C_VEL
LIN {X 0,Y 564.695,Z 389.593,A -85,B 0,C 180,E1 25799.929,E2 25799.929} C_VEL
LIN {X 0,Y 565.793,Z 331.939,A -85,B 0,C 180,E1 25796.523,E2 25796.523} C_VEL
LIN {X 0,Y 566.206,Z 307.048,A -85,B 0,C 180,E1 25795.022,E2 25795.022} C_VEL
LIN {X 0,Y 560.335,Z 293.207,A -85,B 0,C 180,E1 25793.799,E2 25793.799} C_VEL
LIN {X 0,Y 560.268,Z 292.685,A -85,B 0,C 180,E1 25793.54,E2 25793.54} C_VEL
LIN {X 0,Y 560.247,Z 292.687,A -85,B 0,C 180,E1 25790.157,E2 25790.157} C_VEL
LIN {X 0,Y 560.279,Z 292.688,A -85,B 0,C 180,E1 25786.877,E2 25786.877} C_VEL
LIN {X 0,Y 560.252,Z 292.694,A -85,B 0,C 180,E1 25783.569,E2 25783.569} C_VEL
LIN {X 0,Y 560.244,Z 292.697,A -85,B 0,C 180,E1 25780.198,E2 25780.198} C_VEL
LIN {X 0,Y 560.283,Z 292.688,A -85,B 0,C 180,E1 25776.921,E2 25776.921} C_VEL
LIN {X 0,Y 560.233,Z 292.695,A -85,B 0,C 180,E1 25773.714,E2 25773.714} C_VEL
LIN {X 0,Y 560.265,Z 292.698,A -85,B 0,C 180,E1 25770.453,E2 25770.453} C_VEL
LIN {X 0,Y 560.247,Z 292.692,A -85,B 0,C 180,E1 25767.284,E2 25767.284} C_VEL
LIN {X 0,Y 560.228,Z 292.695,A -85,B 0,C 180,E1 25763.97,E2 25763.97} C_VEL
LIN {X 0,Y 560.282,Z 292.695,A -85,B 0,C 180,E1 25760.758,E2 25760.758} C_VEL
LIN {X 0,Y 560.216,Z 292.695,A -85,B 0,C 180,E1 25757.555,E2 25757.555} C_VEL
LIN {X 0,Y 560.25,Z 292.693,A -85,B 0,C 180,E1 25754.293,E2 25754.293} C_VEL
LIN {X 0,Y 560.222,Z 292.697,A -85,B 0,C 180,E1 25751.218,E2 25751.218} C_VEL
LIN {X 0,Y 560.217,Z 292.695,A -85,B 0,C 180,E1 25747.896,E2 25747.896} C_VEL
LIN {X 0,Y 560.248,Z 292.698,A -85,B 0,C 180,E1 25744.811,E2 25744.811} C_VEL
LIN {X 0,Y 560.201,Z 292.697,A -85,B 0,C 180,E1 25741.636,E2 25741.636} C_VEL
LIN {X 0,Y 560.271,Z 292.696,A -85,B 0,C 180,E1 25738.466,E2 25738.466} C_VEL
LIN {X 0,Y 560.198,Z 292.698,A -85,B 0,C 180,E1 25735.29,E2 25735.29} C_VEL
LIN {X 0,Y 560.241,Z 292.692,A -85,B 0,C 180,E1 25732.086,E2 25732.086} C_VEL
LIN {X 0,Y 560.215,Z 292.698,A -85,B 0,C 180,E1 25728.99,E2 25728.99} C_VEL
LIN {X 0,Y 560.215,Z 292.692,A -85,B 0,C 180,E1 25725.636,E2 25725.636} C_VEL
LIN {X 0,Y 560.256,Z 292.699,A -85,B 0,C 180,E1 25722.553,E2 25722.553} C_VEL
LIN {X 0,Y 560.213,Z 292.695,A -85,B 0,C 180,E1 25719.305,E2 25719.305} C_VEL
LIN {X 0,Y 560.282,Z 292.693,A -85,B 0,C 180,E1 25716.313,E2 25716.313} C_VEL
LIN {X 0,Y 559.276,Z 292.812,A -85,B 0,C 180,E1 25715.525,E2 25715.525} C_VEL
LIN {X 0,Y 552.789,Z 293.623,A -85,B 0,C 180,E1 25713.314,E2 25713.314} C_VEL
LIN {X 0,Y 552.299,Z 293.687,A -85,B 0,C 180,E1 25712.738,E2 25712.738} C_VEL
LIN {X 0,Y 552.291,Z 293.683,A -85,B 0,C 180,E1 25709.421,E2 25709.421} C_VEL
LIN {X 0,Y 552.343,Z 293.682,A -85,B 0,C 180,E1 25706.188,E2 25706.188} C_VEL
LIN {X 0,Y 552.293,Z 293.685,A -85,B 0,C 180,E1 25702.925,E2 25702.925} C_VEL
LIN {X 0,Y 552.319,Z 293.681,A -85,B 0,C 180,E1 25699.602,E2 25699.602} C_VEL
LIN {X 0,Y 552.327,Z 293.688,A -85,B 0,C 180,E1 25696.392,E2 25696.392} C_VEL
LIN {X 0,Y 552.3,Z 293.674,A -85,B 0,C 180,E1 25693.038,E2 25693.038} C_VEL
LIN {X 0,Y 552.341,Z 293.675,A -85,B 0,C 180,E1 25689.716,E2 25689.716} C_VEL
LIN {X 0,Y 552.33,Z 293.687,A -85,B 0,C 180,E1 25686.335,E2 25686.335} C_VEL
LIN {X 0,Y 552.311,Z 293.684,A -85,B 0,C 180,E1 25683.017,E2 25683.017} C_VEL
LIN {X 0,Y 552.342,Z 293.683,A -85,B 0,C 180,E1 25679.668,E2 25679.668} C_VEL
LIN {X 0,Y 552.352,Z 293.975,A -85,B 0,C 180,E1 25678.821,E2 25678.821} C_VEL
LIN {X 0,Y 556.072,Z 305.628,A -85,B 0,C 180,E1 25677.406,E2 25677.406} C_VEL
LIN {X 0,Y 555.276,Z 335.267,A -85,B 0,C 180,E1 25674.628,E2 25674.628} C_VEL
LIN {X 0,Y 556.816,Z 344.275,A -85,B 0,C 180,E1 25674.409,E2 25674.409} C_VEL
LIN {X 0,Y 555.686,Z 542.378,A -85,B 0,C 180,E1 25671.669,E2 25671.669} C_VEL
LIN {X 0,Y 555.397,Z 561.24,A -85,B 0,C 180,E1 25671.213,E2 25671.213} C_VEL
LIN {X 0,Y 554.964,Z 579.491,A -85,B 0,C 180,E1 25670.568,E2 25670.568} C_VEL
LIN {X 0,Y 554.492,Z 596.687,A -85,B 0,C 180,E1 25669.755,E2 25669.755} C_VEL
LIN {X 0,Y 553.933,Z 616.269,A -85,B 0,C 180,E1 25668.582,E2 25668.582} C_VEL
LIN {X 0,Y 553.499,Z 632.409,A -85,B 0,C 180,E1 25667.395,E2 25667.395} C_VEL
LIN {X 0,Y 553.09,Z 647.422,A -85,B 0,C 180,E1 25666.056,E2 25666.056} C_VEL
LIN {X 0,Y 552.732,Z 661.164,A -85,B 0,C 180,E1 25664.582,E2 25664.582} C_VEL
LIN {X 0,Y 552.457,Z 672.902,A -85,B 0,C 180,E1 25663.075,E2 25663.075} C_VEL
LIN {X 0,Y 552.23,Z 683.866,A -85,B 0,C 180,E1 25661.382,E2 25661.382} C_VEL
LIN {X 0,Y 552.076,Z 693.318,A -85,B 0,C 180,E1 25659.591,E2 25659.591} C_VEL
LIN {X 0,Y 551.986,Z 700.982,A -85,B 0,C 180,E1 25657.765,E2 25657.765} C_VEL
LIN {X 0,Y 551.932,Z 707.192,A -85,B 0,C 180,E1 25655.822,E2 25655.822} C_VEL
LIN {X 0,Y 551.92,Z 711.605,A -85,B 0,C 180,E1 25653.843,E2 25653.843} C_VEL
LIN {X 0,Y 551.914,Z 714.178,A -85,B 0,C 180,E1 25651.869,E2 25651.869} C_VEL
LIN {X 0,Y 551.916,Z 714.992,A -85,B 0,C 180,E1 25649.896,E2 25649.896} C_VEL
LIN {X 0,Y 551.917,Z 714.065,A -85,B 0,C 180,E1 25647.924,E2 25647.924} C_VEL
LIN {X 0,Y 551.921,Z 711.376,A -85,B 0,C 180,E1 25645.949,E2 25645.949} C_VEL
LIN {X 0,Y 551.937,Z 706.971,A -85,B 0,C 180,E1 25644.011,E2 25644.011} C_VEL
LIN {X 0,Y 551.988,Z 700.76,A -85,B 0,C 180,E1 25642.088,E2 25642.088} C_VEL
LIN {X 0,Y 552.077,Z 693.245,A -85,B 0,C 180,E1 25640.304,E2 25640.304} C_VEL
LIN {X 0,Y 552.231,Z 683.772,A -85,B 0,C 180,E1 25638.512,E2 25638.512} C_VEL
LIN {X 0,Y 552.458,Z 672.783,A -85,B 0,C 180,E1 25636.819,E2 25636.819} C_VEL
LIN {X 0,Y 552.755,Z 660.265,A -85,B 0,C 180,E1 25635.224,E2 25635.224} C_VEL
LIN {X 0,Y 553.124,Z 646.131,A -85,B 0,C 180,E1 25633.729,E2 25633.729} C_VEL
LIN {X 0,Y 553.539,Z 630.846,A -85,B 0,C 180,E1 25632.389,E2 25632.389} C_VEL
LIN {X 0,Y 553.959,Z 615.253,A -85,B 0,C 180,E1 25631.26,E2 25631.26} C_VEL
LIN {X 0,Y 554.497,Z 596.601,A -85,B 0,C 180,E1 25630.151,E2 25630.151} C_VEL
